SPLINE
SPL {X  -146.983, Y  +302.107, Z    +0.000, E1   +74.473, E3 +78846.478}
SPL {X  -146.624, Y  +301.420, Z    +0.000, E1   +73.294, E3 +78856.962}
SPL {X  -144.830, Y  +298.101, Z    +0.000, E1   +72.333, E3 +78866.485}
SPL {X  -140.483, Y  +290.724, Z    +0.000, E1   +71.922, E3 +78873.643}
SPL {X  -136.362, Y  +284.451, Z    +0.000, E1   +71.514, E3 +78879.809}
SPL {X  -132.604, Y  +279.221, Z    +0.000, E1   +70.988, E3 +78885.838}
SPL {X  -129.663, Y  +275.410, Z    +0.000, E1   +70.632, E3 +78889.761}
SPL {X  -127.149, Y  +272.325, Z    +0.000, E1   +70.073, E3 +78894.141}
SPL {X  -123.924, Y  +268.578, Z    +0.000, E1   +70.633, E3 +78893.958}
SPL {X  -115.163, Y  +259.431, Z    +0.000, E1   +74.058, E3 +78885.067}
SPL {X   -55.479, Y  +222.417, Z    +0.000, E1   +56.403, E3 +79070.921}
ENDSPLINE

SPLINE
SPL {X  -130.757, Y  +276.802, Z    +0.000, E1   +58.343, E3 +79226.857}
SPL {X  -154.788, Y  +319.502, Z    +0.000, E1   +45.389, E3 +79231.056}
SPL {X  -161.887, Y  +343.393, Z    +0.000, E1   +32.461, E3 +79231.512}
SPL {X  -164.949, Y  +363.277, Z    +0.000, E1   +17.059, E3 +79230.787}
SPL {X  -165.638, Y  +376.493, Z    +0.000, E1    +4.395, E3 +79230.425}
SPL {X  -165.650, Y  +380.829, Z    +0.000, E1    -0.360, E3 +79229.405}
SPL {X  -165.650, Y  +385.053, Z    +0.000, E1   -10.073, E3 +79228.913}
SPL {X  -165.650, Y  +388.847, Z    +0.000, E1   -19.524, E3 +79228.878}
SPL {X  -165.650, Y  +394.451, Z    +0.000, E1   -33.170, E3 +79228.291}
SPL {X  -165.650, Y  +401.692, Z    +0.000, E1   -47.300, E3 +79228.273}
SPL {X  -165.650, Y  +412.079, Z    +0.000, E1   -62.360, E3 +79226.115}
SPL {X  -165.650, Y  +422.274, Z    +0.000, E1   -68.953, E3 +79226.601}
SPL {X  -165.650, Y  +470.008, Z    +0.000, E1   -77.011, E3 +79234.818}
SPL {X  -161.095, Y  +714.078, Z    +0.000, E1   -78.221, E3 +79310.354}
ENDSPLINE

SPLINE
SPL {X  -163.418, Y  +702.603, Z    +0.000, E1   -74.313, E3 +79347.749}
ENDSPLINE

SPLINE
SPL {X  -160.284, Y  +717.322, Z    +0.000, E1   -73.988, E3 +79359.513}
SPL {X  -156.453, Y  +729.928, Z    +0.000, E1   -73.507, E3 +79371.665}
SPL {X  -152.193, Y  +740.900, Z    +0.000, E1   -73.135, E3 +79381.232}
SPL {X  -148.880, Y  +748.126, Z    +0.000, E1   -72.716, E3 +79389.013}
SPL {X  -145.823, Y  +754.085, Z    +0.000, E1   -72.288, E3 +79395.784}
SPL {X  -141.906, Y  +760.955, Z    +0.000, E1   -72.057, E3 +79401.475}
SPL {X  -138.580, Y  +766.249, Z    +0.000, E1   -71.449, E3 +79408.565}
SPL {X  -134.851, Y  +771.704, Z    +0.000, E1   -71.081, E3 +79413.960}
SPL {X  -131.668, Y  +776.015, Z    +0.000, E1   -70.566, E3 +79419.234}
SPL {X  -127.547, Y  +781.197, Z    +0.000, E1   -70.083, E3 +79424.597}
SPL {X  -118.977, Y  +790.758, Z    +0.000, E1   -71.976, E3 +79422.115}
SPL {X   -54.368, Y  +831.974, Z    +0.000, E1   -57.152, E3 +79573.904}
ENDSPLINE

SPLINE
SPL {X  -111.514, Y  +797.993, Z    +0.000, E1   -63.064, E3 +79760.035}
SPL {X  -140.675, Y  +762.967, Z    +0.000, E1   -56.489, E3 +79765.998}
SPL {X  -155.138, Y  +733.569, Z    +0.000, E1   -46.550, E3 +79768.302}
SPL {X  -161.585, Y  +711.971, Z    +0.000, E1   -34.503, E3 +79767.352}
SPL {X  -164.796, Y  +692.295, Z    +0.000, E1   -19.289, E3 +79767.387}
SPL {X  -165.632, Y  +677.938, Z    +0.000, E1    -5.073, E3 +79766.758}
SPL {X  -165.650, Y  +673.500, Z    +0.000, E1    +0.000, E3 +79765.792}
SPL {X  -165.650, Y  +671.349, Z    +0.000, E1    +4.619, E3 +79765.297}
SPL {X  -165.650, Y  +666.568, Z    +0.000, E1   +16.799, E3 +79765.172}
SPL {X  -165.650, Y  +661.246, Z    +0.000, E1   +30.569, E3 +79764.952}
SPL {X  -165.650, Y  +652.403, Z    +0.000, E1   +48.665, E3 +79764.591}
SPL {X  -165.650, Y  +637.100, Z    +0.000, E1   +69.106, E3 +79760.931}
SPL {X  -165.650, Y  +616.344, Z    +0.000, E1   +74.941, E3 +79764.181}
SPL {X  -165.650, Y  +575.817, Z    +0.000, E1   +77.800, E3 +79773.110}
SPL {X  -161.405, Y  +341.238, Z    +0.000, E1   +76.606, E3 +79864.409}
SPL {X  -146.302, Y  +300.811, Z    +0.000, E1   +78.008, E3 +79865.526}
ENDSPLINE

SPLINE
SPL {X  -147.825, Y  +303.750, Z    +0.000, E1   +76.548, E3 +79879.958}
SPL {X  -148.167, Y  +304.430, Z    +0.000, E1   +75.276, E3 +79892.051}
ENDSPLINE

SPLINE
SPL {X  -146.983, Y  +302.107, Z    +0.000, E1   +74.473, E3 +79900.532}
SPL {X  -146.624, Y  +301.420, Z    +0.000, E1   +73.294, E3 +79911.016}
SPL {X  -144.830, Y  +298.101, Z    +0.000, E1   +72.333, E3 +79920.540}
SPL {X  -140.483, Y  +290.724, Z    +0.000, E1   +71.922, E3 +79927.697}
SPL {X  -136.362, Y  +284.451, Z    +0.000, E1   +71.514, E3 +79933.863}
SPL {X  -132.604, Y  +279.221, Z    +0.000, E1   +70.988, E3 +79939.892}
SPL {X  -129.663, Y  +275.410, Z    +0.000, E1   +70.632, E3 +79943.815}
SPL {X  -127.149, Y  +272.325, Z    +0.000, E1   +70.073, E3 +79948.195}
SPL {X  -123.924, Y  +268.578, Z    +0.000, E1   +70.633, E3 +79948.012}
SPL {X  -115.163, Y  +259.431, Z    +0.000, E1   +74.058, E3 +79939.121}
SPL {X   -55.479, Y  +222.417, Z    +0.000, E1   +56.403, E3 +80124.975}
ENDSPLINE

SPLINE
SPL {X  -130.757, Y  +276.802, Z    +0.000, E1   +58.343, E3 +80280.911}
SPL {X  -154.788, Y  +319.502, Z    +0.000, E1   +45.389, E3 +80285.110}
SPL {X  -161.887, Y  +343.393, Z    +0.000, E1   +32.461, E3 +80285.566}
SPL {X  -164.949, Y  +363.277, Z    +0.000, E1   +17.059, E3 +80284.841}
SPL {X  -165.638, Y  +376.493, Z    +0.000, E1    +4.395, E3 +80284.479}
SPL {X  -165.650, Y  +380.500, Z    +0.000, E1    +0.000, E3 +80283.590}
SPL {X  -165.650, Y  +381.832, Z    +0.000, E1    -2.686, E3 +80283.062}
SPL {X  -165.650, Y  +385.053, Z    +0.000, E1   -10.073, E3 +80282.967}
SPL {X  -165.650, Y  +388.847, Z    +0.000, E1   -19.524, E3 +80282.932}
SPL {X  -165.650, Y  +393.562, Z    +0.000, E1   -31.212, E3 +80282.415}
SPL {X  -165.650, Y  +400.090, Z    +0.000, E1   -44.561, E3 +80282.270}
SPL {X  -165.650, Y  +415.429, Z    +0.000, E1   -64.815, E3 +80280.329}
SPL {X  -165.650, Y  +470.008, Z    +0.000, E1   -77.011, E3 +80288.873}
SPL {X  -160.882, Y  +714.957, Z    +0.000, E1   -77.470, E3 +80372.578}
ENDSPLINE

SPLINE
SPL {X  -163.522, Y  +701.969, Z    +0.000, E1   -74.236, E3 +80402.234}
ENDSPLINE

SPLINE
SPL {X  -160.284, Y  +717.322, Z    +0.000, E1   -73.988, E3 +80413.567}
SPL {X  -156.453, Y  +729.928, Z    +0.000, E1   -73.507, E3 +80425.719}
SPL {X  -152.193, Y  +740.900, Z    +0.000, E1   -73.135, E3 +80435.286}
SPL {X  -148.880, Y  +748.126, Z    +0.000, E1   -72.716, E3 +80443.067}
SPL {X  -144.434, Y  +756.610, Z    +0.000, E1   -72.338, E3 +80450.917}
SPL {X  -141.532, Y  +761.573, Z    +0.000, E1   -71.800, E3 +80457.557}
SPL {X  -138.580, Y  +766.249, Z    +0.000, E1   -71.449, E3 +80462.619}
SPL {X  -134.851, Y  +771.704, Z    +0.000, E1   -71.081, E3 +80468.014}
SPL {X  -131.668, Y  +776.015, Z    +0.000, E1   -70.566, E3 +80473.288}
SPL {X  -128.114, Y  +780.508, Z    +0.000, E1   -70.155, E3 +80477.883}
SPL {X  -123.825, Y  +785.533, Z    +0.000, E1   -70.642, E3 +80478.631}
SPL {X  -111.068, Y  +798.397, Z    +0.000, E1   -72.944, E3 +80476.075}
SPL {X   -54.135, Y  +832.054, Z    +0.000, E1   -56.519, E3 +80652.094}
ENDSPLINE

SPLINE
SPL {X  -119.915, Y  +789.781, Z    +0.000, E1   -62.637, E3 +80819.710}
SPL {X  -140.675, Y  +762.967, Z    +0.000, E1   -56.489, E3 +80820.052}
SPL {X  -155.138, Y  +733.569, Z    +0.000, E1   -46.550, E3 +80822.356}
SPL {X  -161.585, Y  +711.971, Z    +0.000, E1   -34.503, E3 +80821.407}
SPL {X  -164.796, Y  +692.295, Z    +0.000, E1   -19.289, E3 +80821.441}
SPL {X  -165.632, Y  +677.938, Z    +0.000, E1    -5.073, E3 +80820.812}
SPL {X  -165.650, Y  +673.500, Z    +0.000, E1    +0.000, E3 +80819.846}
SPL {X  -165.650, Y  +671.349, Z    +0.000, E1    +4.619, E3 +80819.351}
SPL {X  -165.650, Y  +666.568, Z    +0.000, E1   +16.799, E3 +80819.226}
SPL {X  -165.650, Y  +661.246, Z    +0.000, E1   +30.569, E3 +80819.007}
SPL {X  -165.650, Y  +652.403, Z    +0.000, E1   +48.665, E3 +80818.645}
SPL {X  -165.650, Y  +637.100, Z    +0.000, E1   +69.106, E3 +80814.985}
SPL {X  -165.650, Y  +616.344, Z    +0.000, E1   +74.941, E3 +80818.235}
SPL {X  -165.650, Y  +575.817, Z    +0.000, E1   +77.800, E3 +80827.164}
SPL {X  -161.405, Y  +341.238, Z    +0.000, E1   +76.606, E3 +80918.463}
SPL {X  -146.302, Y  +300.811, Z    +0.000, E1   +78.008, E3 +80919.580}
ENDSPLINE

SPLINE
SPL {X  -147.825, Y  +303.750, Z    +0.000, E1   +76.548, E3 +80934.013}
SPL {X  -148.167, Y  +304.430, Z    +0.000, E1   +75.276, E3 +80946.105}
ENDSPLINE

SPLINE
SPL {X  -146.983, Y  +302.107, Z    +0.000, E1   +74.473, E3 +80954.586}
SPL {X  -146.624, Y  +301.420, Z    +0.000, E1   +73.294, E3 +80965.070}
SPL {X  -144.830, Y  +298.101, Z    +0.000, E1   +72.333, E3 +80974.594}
SPL {X  -140.980, Y  +291.526, Z    +0.000, E1   +72.160, E3 +80979.519}
SPL {X  -137.379, Y  +285.943, Z    +0.000, E1   +71.537, E3 +80986.973}
SPL {X  -133.329, Y  +280.198, Z    +0.000, E1   +71.389, E3 +80991.002}
SPL {X  -130.835, Y  +276.902, Z    +0.000, E1   +70.642, E3 +80996.998}
SPL {X  -127.149, Y  +272.325, Z    +0.000, E1   +70.073, E3 +81002.249}
SPL {X  -123.924, Y  +268.578, Z    +0.000, E1   +70.633, E3 +81002.066}
SPL {X  -115.163, Y  +259.431, Z    +0.000, E1   +74.058, E3 +80993.175}
SPL {X   -55.479, Y  +222.417, Z    +0.000, E1   +56.403, E3 +81179.029}
ENDSPLINE

SPLINE
SPL {X  -130.757, Y  +276.802, Z    +0.000, E1   +58.343, E3 +81334.966}
SPL {X  -154.788, Y  +319.502, Z    +0.000, E1   +45.389, E3 +81339.164}
SPL {X  -161.887, Y  +343.393, Z    +0.000, E1   +32.461, E3 +81339.620}
SPL {X  -164.949, Y  +363.277, Z    +0.000, E1   +17.059, E3 +81338.895}
SPL {X  -165.638, Y  +376.493, Z    +0.000, E1    +4.395, E3 +81338.534}
SPL {X  -165.650, Y  +380.500, Z    +0.000, E1    +0.000, E3 +81337.644}
SPL {X  -165.650, Y  +381.832, Z    +0.000, E1    -2.686, E3 +81337.116}
SPL {X  -165.650, Y  +385.053, Z    +0.000, E1   -10.073, E3 +81337.021}
SPL {X  -165.650, Y  +388.847, Z    +0.000, E1   -19.524, E3 +81336.986}
SPL {X  -165.650, Y  +393.562, Z    +0.000, E1   -31.212, E3 +81336.470}
SPL {X  -165.650, Y  +400.090, Z    +0.000, E1   -44.561, E3 +81336.324}
SPL {X  -165.650, Y  +415.429, Z    +0.000, E1   -64.815, E3 +81334.383}
SPL {X  -165.650, Y  +470.008, Z    +0.000, E1   -77.011, E3 +81342.927}
SPL {X  -160.882, Y  +714.957, Z    +0.000, E1   -77.470, E3 +81426.632}
ENDSPLINE

SPLINE
SPL {X  -164.302, Y  +696.586, Z    +0.000, E1   -74.218, E3 +81453.294}
ENDSPLINE

SPLINE
SPL {X  -160.977, Y  +714.570, Z    +0.000, E1   -74.086, E3 +81465.206}
SPL {X  -156.453, Y  +729.928, Z    +0.000, E1   -73.507, E3 +81479.773}
SPL {X  -152.193, Y  +740.900, Z    +0.000, E1   -73.135, E3 +81489.340}
SPL {X  -148.880, Y  +748.126, Z    +0.000, E1   -72.716, E3 +81497.121}
SPL {X  -144.434, Y  +756.610, Z    +0.000, E1   -72.338, E3 +81504.971}
SPL {X  -141.532, Y  +761.573, Z    +0.000, E1   -71.800, E3 +81511.611}
SPL {X  -138.580, Y  +766.249, Z    +0.000, E1   -71.449, E3 +81516.673}
SPL {X  -134.851, Y  +771.704, Z    +0.000, E1   -71.081, E3 +81522.068}
SPL {X  -131.668, Y  +776.015, Z    +0.000, E1   -70.566, E3 +81527.342}
SPL {X  -128.114, Y  +780.508, Z    +0.000, E1   -70.155, E3 +81531.937}
SPL {X  -125.843, Y  +783.219, Z    +0.000, E1   -69.779, E3 +81535.041}
SPL {X  -118.977, Y  +790.758, Z    +0.000, E1   -71.976, E3 +81530.223}
SPL {X   -54.135, Y  +832.054, Z    +0.000, E1   -56.519, E3 +81706.148}
ENDSPLINE

SPLINE
SPL {X  -119.915, Y  +789.781, Z    +0.000, E1   -62.637, E3 +81873.764}
SPL {X  -140.675, Y  +762.967, Z    +0.000, E1   -56.489, E3 +81874.106}
SPL {X  -155.138, Y  +733.569, Z    +0.000, E1   -46.550, E3 +81876.410}
SPL {X  -161.585, Y  +711.971, Z    +0.000, E1   -34.503, E3 +81875.461}
SPL {X  -164.796, Y  +692.295, Z    +0.000, E1   -19.289, E3 +81875.495}
SPL {X  -165.571, Y  +680.631, Z    +0.000, E1    -7.833, E3 +81874.942}
SPL {X  -165.650, Y  +673.591, Z    +0.000, E1    -0.194, E3 +81873.946}
SPL {X  -165.650, Y  +671.349, Z    +0.000, E1    +4.619, E3 +81873.405}
SPL {X  -165.650, Y  +666.568, Z    +0.000, E1   +16.799, E3 +81873.281}
SPL {X  -165.650, Y  +661.246, Z    +0.000, E1   +30.569, E3 +81873.061}
SPL {X  -165.650, Y  +655.398, Z    +0.000, E1   +43.871, E3 +81872.508}
SPL {X  -165.650, Y  +646.168, Z    +0.000, E1   +58.442, E3 +81871.603}
SPL {X  -165.650, Y  +629.125, Z    +0.000, E1   +72.389, E3 +81869.900}
SPL {X  -165.650, Y  +575.817, Z    +0.000, E1   +77.800, E3 +81881.218}
SPL {X  -161.405, Y  +341.238, Z    +0.000, E1   +76.606, E3 +81972.518}
SPL {X  -146.302, Y  +300.811, Z    +0.000, E1   +78.008, E3 +81973.634}
ENDSPLINE

SPLINE
SPL {X  -147.825, Y  +303.750, Z    +0.000, E1   +76.548, E3 +81988.067}
SPL {X  -148.167, Y  +304.430, Z    +0.000, E1   +75.276, E3 +82000.159}
ENDSPLINE

SPLINE
SPL {X  -146.983, Y  +302.107, Z    +0.000, E1   +74.473, E3 +82008.640}
SPL {X  -146.624, Y  +301.420, Z    +0.000, E1   +73.294, E3 +82019.124}
SPL {X  -144.830, Y  +298.101, Z    +0.000, E1   +72.333, E3 +82028.648}
SPL {X  -140.980, Y  +291.526, Z    +0.000, E1   +72.160, E3 +82033.573}
SPL {X  -137.379, Y  +285.943, Z    +0.000, E1   +71.537, E3 +82041.028}
SPL {X  -133.329, Y  +280.198, Z    +0.000, E1   +71.389, E3 +82045.056}
SPL {X  -130.835, Y  +276.902, Z    +0.000, E1   +70.642, E3 +82051.052}
SPL {X  -127.149, Y  +272.325, Z    +0.000, E1   +70.073, E3 +82056.303}
SPL {X  -123.924, Y  +268.578, Z    +0.000, E1   +70.633, E3 +82056.120}
SPL {X  -115.163, Y  +259.431, Z    +0.000, E1   +74.058, E3 +82047.229}
SPL {X   -55.479, Y  +222.417, Z    +0.000, E1   +56.403, E3 +82233.083}
ENDSPLINE

SPLINE
SPL {X  -130.757, Y  +276.802, Z    +0.000, E1   +58.343, E3 +82389.020}
SPL {X  -154.788, Y  +319.502, Z    +0.000, E1   +45.389, E3 +82393.218}
SPL {X  -161.887, Y  +343.393, Z    +0.000, E1   +32.461, E3 +82393.674}
SPL {X  -164.949, Y  +363.277, Z    +0.000, E1   +17.059, E3 +82392.949}
SPL {X  -165.638, Y  +376.493, Z    +0.000, E1    +4.395, E3 +82392.588}
SPL {X  -165.650, Y  +380.500, Z    +0.000, E1    +0.000, E3 +82391.698}
SPL {X  -165.650, Y  +381.832, Z    +0.000, E1    -2.686, E3 +82391.170}
SPL {X  -165.650, Y  +385.053, Z    +0.000, E1   -10.073, E3 +82391.075}
SPL {X  -165.650, Y  +388.847, Z    +0.000, E1   -19.524, E3 +82391.040}
SPL {X  -165.650, Y  +393.562, Z    +0.000, E1   -31.212, E3 +82390.524}
SPL {X  -165.650, Y  +400.090, Z    +0.000, E1   -44.561, E3 +82390.378}
SPL {X  -165.650, Y  +415.429, Z    +0.000, E1   -64.815, E3 +82388.437}
SPL {X  -165.650, Y  +470.008, Z    +0.000, E1   -77.011, E3 +82396.981}
SPL {X  -160.882, Y  +714.957, Z    +0.000, E1   -77.470, E3 +82480.687}
ENDSPLINE

SPLINE
SPL {X  -164.302, Y  +696.586, Z    +0.000, E1   -74.218, E3 +82507.348}
ENDSPLINE

SPLINE
SPL {X  -160.977, Y  +714.570, Z    +0.000, E1   -74.086, E3 +82519.260}
SPL {X  -156.453, Y  +729.928, Z    +0.000, E1   -73.507, E3 +82533.827}
SPL {X  -152.193, Y  +740.900, Z    +0.000, E1   -73.135, E3 +82543.394}
SPL {X  -148.880, Y  +748.126, Z    +0.000, E1   -72.716, E3 +82551.175}
SPL {X  -144.434, Y  +756.610, Z    +0.000, E1   -72.338, E3 +82559.025}
SPL {X  -141.532, Y  +761.573, Z    +0.000, E1   -71.800, E3 +82565.665}
SPL {X  -138.580, Y  +766.249, Z    +0.000, E1   -71.449, E3 +82570.727}
SPL {X  -134.851, Y  +771.704, Z    +0.000, E1   -71.081, E3 +82576.122}
SPL {X  -131.668, Y  +776.015, Z    +0.000, E1   -70.566, E3 +82581.396}
SPL {X  -128.114, Y  +780.508, Z    +0.000, E1   -70.155, E3 +82585.991}
SPL {X  -125.843, Y  +783.219, Z    +0.000, E1   -69.779, E3 +82589.095}
SPL {X  -118.977, Y  +790.758, Z    +0.000, E1   -71.976, E3 +82584.277}
SPL {X   -54.135, Y  +832.054, Z    +0.000, E1   -56.519, E3 +82760.202}
ENDSPLINE

SPLINE
SPL {X  -119.915, Y  +789.781, Z    +0.000, E1   -62.637, E3 +82927.818}
SPL {X  -140.675, Y  +762.967, Z    +0.000, E1   -56.489, E3 +82928.160}
SPL {X  -155.138, Y  +733.569, Z    +0.000, E1   -46.550, E3 +82930.464}
SPL {X  -161.585, Y  +711.971, Z    +0.000, E1   -34.503, E3 +82929.515}
SPL {X  -164.796, Y  +692.295, Z    +0.000, E1   -19.289, E3 +82929.549}
SPL {X  -165.571, Y  +680.631, Z    +0.000, E1    -7.833, E3 +82928.996}
SPL {X  -165.650, Y  +673.591, Z    +0.000, E1    -0.194, E3 +82928.000}
SPL {X  -165.650, Y  +671.349, Z    +0.000, E1    +4.619, E3 +82927.459}
SPL {X  -165.650, Y  +666.568, Z    +0.000, E1   +16.799, E3 +82927.335}
SPL {X  -165.650, Y  +661.246, Z    +0.000, E1   +30.569, E3 +82927.115}
SPL {X  -165.650, Y  +655.398, Z    +0.000, E1   +43.871, E3 +82926.562}
SPL {X  -165.650, Y  +646.168, Z    +0.000, E1   +58.442, E3 +82925.657}
SPL {X  -165.650, Y  +629.125, Z    +0.000, E1   +72.389, E3 +82923.954}
SPL {X  -165.650, Y  +575.817, Z    +0.000, E1   +77.800, E3 +82935.272}
SPL {X  -161.405, Y  +341.238, Z    +0.000, E1   +76.606, E3 +83026.572}
SPL {X  -146.302, Y  +300.811, Z    +0.000, E1   +78.008, E3 +83027.688}
ENDSPLINE

SPLINE
SPL {X  -147.825, Y  +303.750, Z    +0.000, E1   +76.548, E3 +83042.121}
SPL {X  -148.167, Y  +304.430, Z    +0.000, E1   +75.276, E3 +83054.214}
ENDSPLINE

SPLINE
SPL {X  -146.983, Y  +302.107, Z    +0.000, E1   +74.473, E3 +83062.694}
SPL {X  -146.624, Y  +301.420, Z    +0.000, E1   +73.294, E3 +83073.178}
SPL {X  -144.830, Y  +298.101, Z    +0.000, E1   +72.333, E3 +83082.702}
SPL {X  -140.980, Y  +291.526, Z    +0.000, E1   +72.160, E3 +83087.627}
SPL {X  -137.379, Y  +285.943, Z    +0.000, E1   +71.537, E3 +83095.082}
SPL {X  -133.329, Y  +280.198, Z    +0.000, E1   +71.389, E3 +83099.110}
SPL {X  -130.835, Y  +276.902, Z    +0.000, E1   +70.642, E3 +83105.106}
SPL {X  -127.149, Y  +272.325, Z    +0.000, E1   +70.073, E3 +83110.358}
SPL {X  -123.924, Y  +268.578, Z    +0.000, E1   +70.633, E3 +83110.174}
SPL {X  -115.163, Y  +259.431, Z    +0.000, E1   +74.058, E3 +83101.284}
SPL {X   -55.479, Y  +222.417, Z    +0.000, E1   +56.403, E3 +83287.137}
ENDSPLINE

SPLINE
SPL {X  -130.757, Y  +276.802, Z    +0.000, E1   +58.343, E3 +83443.074}
SPL {X  -154.788, Y  +319.502, Z    +0.000, E1   +45.389, E3 +83447.272}
SPL {X  -161.887, Y  +343.393, Z    +0.000, E1   +32.461, E3 +83447.728}
SPL {X  -164.949, Y  +363.277, Z    +0.000, E1   +17.059, E3 +83447.003}
SPL {X  -165.638, Y  +376.493, Z    +0.000, E1    +4.395, E3 +83446.642}
SPL {X  -165.650, Y  +380.500, Z    +0.000, E1    +0.000, E3 +83445.752}
SPL {X  -165.650, Y  +381.832, Z    +0.000, E1    -2.686, E3 +83445.224}
SPL {X  -165.650, Y  +385.053, Z    +0.000, E1   -10.073, E3 +83445.129}
SPL {X  -165.650, Y  +388.847, Z    +0.000, E1   -19.524, E3 +83445.094}
SPL {X  -165.650, Y  +393.562, Z    +0.000, E1   -31.212, E3 +83444.578}
SPL {X  -165.650, Y  +400.090, Z    +0.000, E1   -44.561, E3 +83444.432}
SPL {X  -165.650, Y  +415.429, Z    +0.000, E1   -64.815, E3 +83442.491}
SPL {X  -165.650, Y  +470.008, Z    +0.000, E1   -77.011, E3 +83451.035}
SPL {X  -160.882, Y  +714.957, Z    +0.000, E1   -77.470, E3 +83534.741}
ENDSPLINE

SPLINE
SPL {X  -164.302, Y  +696.586, Z    +0.000, E1   -74.218, E3 +83561.403}
ENDSPLINE

SPLINE
SPL {X  -160.977, Y  +714.570, Z    +0.000, E1   -74.086, E3 +83573.314}
SPL {X  -156.453, Y  +729.928, Z    +0.000, E1   -73.507, E3 +83587.881}
SPL {X  -152.193, Y  +740.900, Z    +0.000, E1   -73.135, E3 +83597.448}
SPL {X  -148.880, Y  +748.126, Z    +0.000, E1   -72.716, E3 +83605.229}
SPL {X  -144.434, Y  +756.610, Z    +0.000, E1   -72.338, E3 +83613.079}
SPL {X  -141.532, Y  +761.573, Z    +0.000, E1   -71.800, E3 +83619.719}
SPL {X  -138.580, Y  +766.249, Z    +0.000, E1   -71.449, E3 +83624.781}
SPL {X  -134.851, Y  +771.704, Z    +0.000, E1   -71.081, E3 +83630.176}
SPL {X  -131.668, Y  +776.015, Z    +0.000, E1   -70.566, E3 +83635.450}
SPL {X  -128.114, Y  +780.508, Z    +0.000, E1   -70.155, E3 +83640.045}
SPL {X  -125.843, Y  +783.219, Z    +0.000, E1   -69.779, E3 +83643.149}
SPL {X  -118.977, Y  +790.758, Z    +0.000, E1   -71.976, E3 +83638.331}
SPL {X   -54.135, Y  +832.054, Z    +0.000, E1   -56.519, E3 +83814.256}
ENDSPLINE

SPLINE
SPL {X  -119.915, Y  +789.781, Z    +0.000, E1   -62.637, E3 +83981.872}
SPL {X  -140.675, Y  +762.967, Z    +0.000, E1   -56.489, E3 +83982.214}
SPL {X  -155.138, Y  +733.569, Z    +0.000, E1   -46.550, E3 +83984.519}
SPL {X  -161.585, Y  +711.971, Z    +0.000, E1   -34.503, E3 +83983.569}
SPL {X  -164.796, Y  +692.295, Z    +0.000, E1   -19.289, E3 +83983.603}
SPL {X  -165.571, Y  +680.631, Z    +0.000, E1    -7.833, E3 +83983.050}
SPL {X  -165.650, Y  +673.591, Z    +0.000, E1    -0.194, E3 +83982.054}
SPL {X  -165.650, Y  +671.349, Z    +0.000, E1    +4.619, E3 +83981.513}
SPL {X  -165.650, Y  +666.568, Z    +0.000, E1   +16.799, E3 +83981.389}
SPL {X  -165.650, Y  +661.246, Z    +0.000, E1   +30.569, E3 +83981.169}
SPL {X  -165.650, Y  +655.398, Z    +0.000, E1   +43.871, E3 +83980.616}
SPL {X  -165.650, Y  +646.168, Z    +0.000, E1   +58.442, E3 +83979.711}
SPL {X  -165.650, Y  +629.125, Z    +0.000, E1   +72.389, E3 +83978.008}
SPL {X  -165.650, Y  +575.817, Z    +0.000, E1   +77.800, E3 +83989.326}
SPL {X  -161.405, Y  +341.238, Z    +0.000, E1   +76.606, E3 +84080.626}
SPL {X  -146.302, Y  +300.811, Z    +0.000, E1   +78.008, E3 +84081.742}
ENDSPLINE

SPLINE
SPL {X  -147.825, Y  +303.750, Z    +0.000, E1   +76.548, E3 +84096.175}
SPL {X  -148.167, Y  +304.430, Z    +0.000, E1   +75.276, E3 +84108.268}
ENDSPLINE

SPLINE
SPL {X  -146.983, Y  +302.107, Z    +0.000, E1   +74.473, E3 +84116.748}
SPL {X  -146.624, Y  +301.420, Z    +0.000, E1   +73.294, E3 +84127.232}
SPL {X  -144.830, Y  +298.101, Z    +0.000, E1   +72.333, E3 +84136.756}
SPL {X  -140.980, Y  +291.526, Z    +0.000, E1   +72.160, E3 +84141.681}
SPL {X  -137.379, Y  +285.943, Z    +0.000, E1   +71.537, E3 +84149.136}
SPL {X  -133.329, Y  +280.198, Z    +0.000, E1   +71.389, E3 +84153.164}
SPL {X  -130.835, Y  +276.902, Z    +0.000, E1   +70.642, E3 +84159.160}
SPL {X  -127.149, Y  +272.325, Z    +0.000, E1   +70.073, E3 +84164.412}
SPL {X  -123.924, Y  +268.578, Z    +0.000, E1   +70.633, E3 +84164.228}
SPL {X  -115.163, Y  +259.431, Z    +0.000, E1   +74.058, E3 +84155.338}
SPL {X   -55.479, Y  +222.417, Z    +0.000, E1   +56.403, E3 +84341.191}
ENDSPLINE

SPLINE
SPL {X  -130.757, Y  +276.802, Z    +0.000, E1   +58.343, E3 +84497.128}
SPL {X  -154.788, Y  +319.502, Z    +0.000, E1   +45.389, E3 +84501.326}
SPL {X  -161.887, Y  +343.393, Z    +0.000, E1   +32.461, E3 +84501.782}
SPL {X  -164.949, Y  +363.277, Z    +0.000, E1   +17.059, E3 +84501.057}
SPL {X  -165.638, Y  +376.493, Z    +0.000, E1    +4.395, E3 +84500.696}
SPL {X  -165.650, Y  +380.500, Z    +0.000, E1    +0.000, E3 +84499.806}
SPL {X  -165.650, Y  +381.832, Z    +0.000, E1    -2.686, E3 +84499.278}
SPL {X  -165.650, Y  +385.053, Z    +0.000, E1   -10.073, E3 +84499.183}
SPL {X  -165.650, Y  +388.847, Z    +0.000, E1   -19.524, E3 +84499.148}
SPL {X  -165.650, Y  +393.562, Z    +0.000, E1   -31.212, E3 +84498.632}
SPL {X  -165.650, Y  +400.090, Z    +0.000, E1   -44.561, E3 +84498.486}
SPL {X  -165.650, Y  +415.429, Z    +0.000, E1   -64.815, E3 +84496.545}
SPL {X  -165.650, Y  +470.008, Z    +0.000, E1   -77.011, E3 +84505.089}
SPL {X  -160.882, Y  +714.957, Z    +0.000, E1   -77.470, E3 +84588.795}
ENDSPLINE

SPLINE
SPL {X  -164.302, Y  +696.586, Z    +0.000, E1   -74.218, E3 +84615.457}
ENDSPLINE

SPLINE
SPL {X  -160.977, Y  +714.570, Z    +0.000, E1   -74.086, E3 +84627.368}
SPL {X  -156.453, Y  +729.928, Z    +0.000, E1   -73.507, E3 +84641.935}
SPL {X  -152.193, Y  +740.900, Z    +0.000, E1   -73.135, E3 +84651.502}
SPL {X  -148.880, Y  +748.126, Z    +0.000, E1   -72.716, E3 +84659.283}
SPL {X  -144.434, Y  +756.610, Z    +0.000, E1   -72.338, E3 +84667.133}
SPL {X  -141.532, Y  +761.573, Z    +0.000, E1   -71.800, E3 +84673.773}
SPL {X  -138.580, Y  +766.249, Z    +0.000, E1   -71.449, E3 +84678.835}
SPL {X  -134.851, Y  +771.704, Z    +0.000, E1   -71.081, E3 +84684.230}
SPL {X  -130.513, Y  +777.511, Z    +0.000, E1   -70.561, E3 +84690.413}
SPL {X  -127.002, Y  +781.850, Z    +0.000, E1   -69.819, E3 +84696.268}
SPL {X  -118.977, Y  +790.758, Z    +0.000, E1   -71.976, E3 +84692.385}
SPL {X   -54.368, Y  +831.974, Z    +0.000, E1   -57.152, E3 +84844.174}
ENDSPLINE

SPLINE
SPL {X  -111.514, Y  +797.993, Z    +0.000, E1   -63.064, E3 +85030.305}
SPL {X  -140.675, Y  +762.967, Z    +0.000, E1   -56.489, E3 +85036.268}
SPL {X  -155.138, Y  +733.569, Z    +0.000, E1   -46.550, E3 +85038.573}
SPL {X  -162.699, Y  +706.626, Z    +0.000, E1   -30.890, E3 +85037.614}
SPL {X  -165.076, Y  +689.274, Z    +0.000, E1   -16.447, E3 +85037.702}
SPL {X  -165.632, Y  +677.938, Z    +0.000, E1    -5.073, E3 +85037.028}
SPL {X  -165.650, Y  +673.500, Z    +0.000, E1    +0.000, E3 +85036.063}
SPL {X  -165.650, Y  +671.349, Z    +0.000, E1    +4.619, E3 +85035.567}
SPL {X  -165.650, Y  +666.568, Z    +0.000, E1   +16.799, E3 +85035.443}
SPL {X  -165.650, Y  +661.246, Z    +0.000, E1   +30.569, E3 +85035.223}
SPL {X  -165.650, Y  +652.403, Z    +0.000, E1   +48.665, E3 +85034.861}
SPL {X  -165.650, Y  +637.100, Z    +0.000, E1   +69.106, E3 +85031.201}
SPL {X  -165.650, Y  +616.344, Z    +0.000, E1   +74.941, E3 +85034.451}
SPL {X  -165.650, Y  +575.817, Z    +0.000, E1   +77.800, E3 +85043.380}
SPL {X  -161.405, Y  +341.238, Z    +0.000, E1   +76.606, E3 +85134.680}
SPL {X  -146.302, Y  +300.811, Z    +0.000, E1   +78.008, E3 +85135.797}
ENDSPLINE

SPLINE
SPL {X  -147.825, Y  +303.750, Z    +0.000, E1   +76.548, E3 +85150.229}
SPL {X  -148.167, Y  +304.430, Z    +0.000, E1   +75.276, E3 +85162.322}
ENDSPLINE

SPLINE
SPL {X  -146.983, Y  +302.107, Z    +0.000, E1   +74.473, E3 +85170.802}
SPL {X  -146.624, Y  +301.420, Z    +0.000, E1   +73.294, E3 +85181.286}
SPL {X  -144.830, Y  +298.101, Z    +0.000, E1   +72.333, E3 +85190.810}
SPL {X  -140.980, Y  +291.526, Z    +0.000, E1   +72.160, E3 +85195.735}
SPL {X  -138.254, Y  +287.254, Z    +0.000, E1   +71.707, E3 +85201.221}
SPL {X  -134.627, Y  +281.983, Z    +0.000, E1   +71.294, E3 +85206.746}
SPL {X  -132.106, Y  +278.560, Z    +0.000, E1   +70.638, E3 +85212.269}
SPL {X  -129.663, Y  +275.410, Z    +0.000, E1   +70.632, E3 +85214.086}
SPL {X  -127.149, Y  +272.325, Z    +0.000, E1   +70.073, E3 +85218.466}
SPL {X  -123.924, Y  +268.578, Z    +0.000, E1   +70.633, E3 +85218.282}
SPL {X  -115.163, Y  +259.431, Z    +0.000, E1   +74.058, E3 +85209.392}
SPL {X   -55.479, Y  +222.417, Z    +0.000, E1   +56.403, E3 +85395.245}
ENDSPLINE

SPLINE
SPL {X  -130.757, Y  +276.802, Z    +0.000, E1   +58.343, E3 +85551.182}
SPL {X  -157.227, Y  +326.349, Z    +0.000, E1   +42.092, E3 +85554.827}
SPL {X  -163.771, Y  +353.623, Z    +0.000, E1   +25.144, E3 +85556.040}
SPL {X  -165.462, Y  +370.602, Z    +0.000, E1   +10.342, E3 +85554.990}
SPL {X  -165.650, Y  +380.752, Z    +0.000, E1    -0.182, E3 +85553.770}
SPL {X  -165.650, Y  +385.053, Z    +0.000, E1   -10.073, E3 +85553.237}
SPL {X  -165.650, Y  +388.847, Z    +0.000, E1   -19.524, E3 +85553.202}
SPL {X  -165.650, Y  +393.562, Z    +0.000, E1   -31.212, E3 +85552.686}
SPL {X  -165.650, Y  +400.090, Z    +0.000, E1   -44.561, E3 +85552.540}
SPL {X  -165.650, Y  +415.429, Z    +0.000, E1   -64.815, E3 +85550.599}
SPL {X  -165.650, Y  +460.635, Z    +0.000, E1   -76.744, E3 +85556.496}
SPL {X  -165.650, Y  +476.745, Z    +0.000, E1   -77.150, E3 +85561.048}
SPL {X  -161.095, Y  +714.078, Z    +0.000, E1   -78.221, E3 +85634.678}
ENDSPLINE

SPLINE
SPL {X  -163.418, Y  +702.603, Z    +0.000, E1   -74.313, E3 +85672.074}
ENDSPLINE

SPLINE
SPL {X  -160.284, Y  +717.322, Z    +0.000, E1   -73.988, E3 +85683.837}
SPL {X  -156.453, Y  +729.928, Z    +0.000, E1   -73.507, E3 +85695.989}
SPL {X  -152.193, Y  +740.900, Z    +0.000, E1   -73.135, E3 +85705.556}
SPL {X  -148.880, Y  +748.126, Z    +0.000, E1   -72.716, E3 +85713.337}
SPL {X  -144.434, Y  +756.610, Z    +0.000, E1   -72.338, E3 +85721.187}
SPL {X  -141.532, Y  +761.573, Z    +0.000, E1   -71.800, E3 +85727.827}
SPL {X  -138.580, Y  +766.249, Z    +0.000, E1   -71.449, E3 +85732.889}
SPL {X  -134.851, Y  +771.704, Z    +0.000, E1   -71.081, E3 +85738.284}
SPL {X  -130.513, Y  +777.511, Z    +0.000, E1   -70.561, E3 +85744.467}
SPL {X  -127.002, Y  +781.850, Z    +0.000, E1   -69.819, E3 +85750.322}
SPL {X  -121.778, Y  +787.794, Z    +0.000, E1   -71.623, E3 +85746.370}
SPL {X  -111.068, Y  +798.397, Z    +0.000, E1   -72.944, E3 +85746.346}
SPL {X   -54.368, Y  +831.974, Z    +0.000, E1   -57.152, E3 +85898.228}
ENDSPLINE

SPLINE
SPL {X  -111.514, Y  +797.993, Z    +0.000, E1   -63.064, E3 +86084.359}
SPL {X  -140.675, Y  +762.967, Z    +0.000, E1   -56.489, E3 +86090.322}
SPL {X  -155.138, Y  +733.569, Z    +0.000, E1   -46.550, E3 +86092.627}
SPL {X  -162.699, Y  +706.626, Z    +0.000, E1   -30.890, E3 +86091.668}
SPL {X  -165.420, Y  +684.230, Z    +0.000, E1   -11.665, E3 +86091.419}
SPL {X  -165.650, Y  +673.591, Z    +0.000, E1    -0.194, E3 +86090.162}
SPL {X  -165.650, Y  +671.349, Z    +0.000, E1    +4.619, E3 +86089.621}
SPL {X  -165.650, Y  +666.568, Z    +0.000, E1   +16.799, E3 +86089.497}
SPL {X  -165.650, Y  +661.246, Z    +0.000, E1   +30.569, E3 +86089.277}
SPL {X  -165.650, Y  +655.398, Z    +0.000, E1   +43.871, E3 +86088.724}
SPL {X  -165.650, Y  +648.742, Z    +0.000, E1   +53.940, E3 +86089.148}
SPL {X  -165.650, Y  +637.100, Z    +0.000, E1   +69.106, E3 +86085.255}
SPL {X  -165.650, Y  +616.344, Z    +0.000, E1   +74.941, E3 +86088.505}
SPL {X  -165.650, Y  +575.817, Z    +0.000, E1   +77.800, E3 +86097.434}
SPL {X  -161.405, Y  +341.238, Z    +0.000, E1   +76.606, E3 +86188.734}
SPL {X  -146.302, Y  +300.811, Z    +0.000, E1   +78.008, E3 +86189.851}
ENDSPLINE

SPLINE
SPL {X  -147.825, Y  +303.750, Z    +0.000, E1   +76.548, E3 +86204.283}
SPL {X  -148.167, Y  +304.430, Z    +0.000, E1   +75.276, E3 +86216.376}
ENDSPLINE

SPLINE
SPL {X  -146.983, Y  +302.107, Z    +0.000, E1   +74.473, E3 +86224.856}
SPL {X  -146.624, Y  +301.420, Z    +0.000, E1   +73.294, E3 +86235.340}
SPL {X  -144.830, Y  +298.101, Z    +0.000, E1   +72.333, E3 +86244.864}
SPL {X  -140.980, Y  +291.526, Z    +0.000, E1   +72.160, E3 +86249.789}
SPL {X  -137.379, Y  +285.943, Z    +0.000, E1   +71.537, E3 +86257.244}
SPL {X  -133.329, Y  +280.198, Z    +0.000, E1   +71.389, E3 +86261.272}
SPL {X  -130.835, Y  +276.902, Z    +0.000, E1   +70.642, E3 +86267.268}
SPL {X  -127.149, Y  +272.325, Z    +0.000, E1   +70.073, E3 +86272.520}
SPL {X  -123.924, Y  +268.578, Z    +0.000, E1   +70.633, E3 +86272.336}
SPL {X  -115.163, Y  +259.431, Z    +0.000, E1   +74.058, E3 +86263.446}
SPL {X   -55.479, Y  +222.417, Z    +0.000, E1   +56.403, E3 +86449.299}
ENDSPLINE

SPLINE
SPL {X  -130.757, Y  +276.802, Z    +0.000, E1   +58.343, E3 +86605.236}
SPL {X  -157.227, Y  +326.349, Z    +0.000, E1   +42.092, E3 +86608.881}
SPL {X  -163.771, Y  +353.623, Z    +0.000, E1   +25.144, E3 +86610.094}
SPL {X  -165.171, Y  +365.918, Z    +0.000, E1   +14.637, E3 +86609.308}
SPL {X  -165.638, Y  +376.493, Z    +0.000, E1    +4.395, E3 +86608.804}
SPL {X  -165.650, Y  +380.500, Z    +0.000, E1    +0.000, E3 +86607.914}
SPL {X  -165.650, Y  +381.832, Z    +0.000, E1    -2.686, E3 +86607.386}
SPL {X  -165.650, Y  +385.053, Z    +0.000, E1   -10.073, E3 +86607.291}
SPL {X  -165.650, Y  +388.847, Z    +0.000, E1   -19.524, E3 +86607.256}
SPL {X  -165.650, Y  +393.562, Z    +0.000, E1   -31.212, E3 +86606.740}
SPL {X  -165.650, Y  +400.090, Z    +0.000, E1   -44.561, E3 +86606.594}
SPL {X  -165.650, Y  +415.429, Z    +0.000, E1   -64.815, E3 +86604.653}
SPL {X  -165.650, Y  +470.008, Z    +0.000, E1   -77.011, E3 +86613.197}
SPL {X  -160.882, Y  +714.957, Z    +0.000, E1   -77.470, E3 +86696.903}
ENDSPLINE

SPLINE
SPL {X  -164.302, Y  +696.586, Z    +0.000, E1   -74.218, E3 +86723.565}
ENDSPLINE

SPLINE
SPL {X  -160.977, Y  +714.570, Z    +0.000, E1   -74.086, E3 +86735.476}
SPL {X  -156.453, Y  +729.928, Z    +0.000, E1   -73.507, E3 +86750.044}
SPL {X  -152.193, Y  +740.900, Z    +0.000, E1   -73.135, E3 +86759.610}
SPL {X  -148.880, Y  +748.126, Z    +0.000, E1   -72.716, E3 +86767.391}
SPL {X  -145.823, Y  +754.085, Z    +0.000, E1   -72.288, E3 +86774.163}
SPL {X  -141.906, Y  +760.955, Z    +0.000, E1   -72.057, E3 +86779.853}
SPL {X  -138.580, Y  +766.249, Z    +0.000, E1   -71.449, E3 +86786.943}
SPL {X  -134.851, Y  +771.704, Z    +0.000, E1   -71.081, E3 +86792.338}
SPL {X  -131.668, Y  +776.015, Z    +0.000, E1   -70.566, E3 +86797.612}
SPL {X  -127.547, Y  +781.197, Z    +0.000, E1   -70.083, E3 +86802.976}
SPL {X  -118.977, Y  +790.758, Z    +0.000, E1   -71.976, E3 +86800.493}
SPL {X   -54.135, Y  +832.054, Z    +0.000, E1   -56.519, E3 +86976.419}
ENDSPLINE

SPLINE
SPL {X  -119.915, Y  +789.781, Z    +0.000, E1   -62.637, E3 +87144.034}
SPL {X  -140.675, Y  +762.967, Z    +0.000, E1   -56.489, E3 +87144.376}
SPL {X  -155.138, Y  +733.569, Z    +0.000, E1   -46.550, E3 +87146.681}
SPL {X  -161.585, Y  +711.971, Z    +0.000, E1   -34.503, E3 +87145.731}
SPL {X  -164.796, Y  +692.295, Z    +0.000, E1   -19.289, E3 +87145.765}
SPL {X  -165.632, Y  +677.938, Z    +0.000, E1    -5.073, E3 +87145.136}
SPL {X  -165.650, Y  +673.500, Z    +0.000, E1    +0.000, E3 +87144.171}
SPL {X  -165.650, Y  +671.349, Z    +0.000, E1    +4.619, E3 +87143.675}
SPL {X  -165.650, Y  +666.568, Z    +0.000, E1   +16.799, E3 +87143.551}
SPL {X  -165.650, Y  +661.246, Z    +0.000, E1   +30.569, E3 +87143.331}
SPL {X  -165.650, Y  +652.403, Z    +0.000, E1   +48.665, E3 +87142.969}
SPL {X  -165.650, Y  +637.100, Z    +0.000, E1   +69.106, E3 +87139.309}
SPL {X  -165.650, Y  +616.344, Z    +0.000, E1   +74.941, E3 +87142.559}
SPL {X  -165.650, Y  +575.817, Z    +0.000, E1   +77.800, E3 +87151.488}
SPL {X  -161.405, Y  +341.238, Z    +0.000, E1   +76.606, E3 +87242.788}
SPL {X  -146.302, Y  +300.811, Z    +0.000, E1   +78.008, E3 +87243.905}
ENDSPLINE

SPLINE
SPL {X  -147.825, Y  +303.750, Z    +0.000, E1   +76.548, E3 +87258.337}
SPL {X  -148.167, Y  +304.430, Z    +0.000, E1   +75.276, E3 +87270.430}
ENDSPLINE

SPLINE
SPL {X  -146.983, Y  +302.107, Z    +0.000, E1   +74.473, E3 +87278.910}
SPL {X  -146.624, Y  +301.420, Z    +0.000, E1   +73.294, E3 +87289.394}
SPL {X  -144.830, Y  +298.101, Z    +0.000, E1   +72.333, E3 +87298.918}
SPL {X  -140.980, Y  +291.526, Z    +0.000, E1   +72.160, E3 +87303.843}
SPL {X  -137.379, Y  +285.943, Z    +0.000, E1   +71.537, E3 +87311.298}
SPL {X  -133.329, Y  +280.198, Z    +0.000, E1   +71.389, E3 +87315.326}
SPL {X  -130.835, Y  +276.902, Z    +0.000, E1   +70.642, E3 +87321.322}
SPL {X  -127.149, Y  +272.325, Z    +0.000, E1   +70.073, E3 +87326.574}
SPL {X  -123.924, Y  +268.578, Z    +0.000, E1   +70.633, E3 +87326.390}
SPL {X  -115.163, Y  +259.431, Z    +0.000, E1   +74.058, E3 +87317.500}
SPL {X   -55.479, Y  +222.417, Z    +0.000, E1   +56.403, E3 +87503.354}
ENDSPLINE

SPLINE
SPL {X  -130.757, Y  +276.802, Z    +0.000, E1   +58.343, E3 +87659.290}
SPL {X  -157.227, Y  +326.349, Z    +0.000, E1   +42.092, E3 +87662.936}
SPL {X  -163.771, Y  +353.623, Z    +0.000, E1   +25.144, E3 +87664.148}
SPL {X  -165.171, Y  +365.918, Z    +0.000, E1   +14.637, E3 +87663.362}
SPL {X  -165.638, Y  +376.493, Z    +0.000, E1    +4.395, E3 +87662.858}
SPL {X  -165.650, Y  +380.500, Z    +0.000, E1    +0.000, E3 +87661.968}
SPL {X  -165.650, Y  +381.832, Z    +0.000, E1    -2.686, E3 +87661.440}
SPL {X  -165.650, Y  +385.053, Z    +0.000, E1   -10.073, E3 +87661.345}
SPL {X  -165.650, Y  +388.847, Z    +0.000, E1   -19.524, E3 +87661.310}
SPL {X  -165.650, Y  +393.562, Z    +0.000, E1   -31.212, E3 +87660.794}
SPL {X  -165.650, Y  +400.090, Z    +0.000, E1   -44.561, E3 +87660.648}
SPL {X  -165.650, Y  +415.429, Z    +0.000, E1   -64.815, E3 +87658.707}
SPL {X  -165.650, Y  +470.008, Z    +0.000, E1   -77.011, E3 +87667.251}
SPL {X  -160.882, Y  +714.957, Z    +0.000, E1   -77.470, E3 +87750.957}
ENDSPLINE

SPLINE
SPL {X  -164.302, Y  +696.586, Z    +0.000, E1   -74.218, E3 +87777.619}
ENDSPLINE

SPLINE
SPL {X  -160.977, Y  +714.570, Z    +0.000, E1   -74.086, E3 +87789.530}
SPL {X  -156.453, Y  +729.928, Z    +0.000, E1   -73.507, E3 +87804.098}
SPL {X  -152.193, Y  +740.900, Z    +0.000, E1   -73.135, E3 +87813.664}
SPL {X  -148.880, Y  +748.126, Z    +0.000, E1   -72.716, E3 +87821.445}
SPL {X  -145.823, Y  +754.085, Z    +0.000, E1   -72.288, E3 +87828.217}
SPL {X  -141.906, Y  +760.955, Z    +0.000, E1   -72.057, E3 +87833.907}
SPL {X  -138.580, Y  +766.249, Z    +0.000, E1   -71.449, E3 +87840.997}
SPL {X  -134.851, Y  +771.704, Z    +0.000, E1   -71.081, E3 +87846.392}
SPL {X  -131.668, Y  +776.015, Z    +0.000, E1   -70.566, E3 +87851.666}
SPL {X  -127.547, Y  +781.197, Z    +0.000, E1   -70.083, E3 +87857.030}
SPL {X  -118.977, Y  +790.758, Z    +0.000, E1   -71.976, E3 +87854.547}
SPL {X   -54.368, Y  +831.974, Z    +0.000, E1   -57.152, E3 +88006.336}
ENDSPLINE

SPLINE
SPL {X  -111.514, Y  +797.993, Z    +0.000, E1   -63.064, E3 +88192.467}
SPL {X  -140.675, Y  +762.967, Z    +0.000, E1   -56.489, E3 +88198.430}
SPL {X  -155.138, Y  +733.569, Z    +0.000, E1   -46.550, E3 +88200.735}
SPL {X  -162.699, Y  +706.626, Z    +0.000, E1   -30.890, E3 +88199.776}
SPL {X  -165.076, Y  +689.274, Z    +0.000, E1   -16.447, E3 +88199.864}
SPL {X  -165.632, Y  +677.938, Z    +0.000, E1    -5.073, E3 +88199.191}
SPL {X  -165.650, Y  +673.297, Z    +0.000, E1    +0.232, E3 +88198.147}
SPL {X  -165.650, Y  +670.223, Z    +0.000, E1    +7.575, E3 +88197.628}
SPL {X  -165.650, Y  +666.568, Z    +0.000, E1   +16.799, E3 +88197.605}
SPL {X  -165.650, Y  +661.246, Z    +0.000, E1   +30.569, E3 +88197.385}
SPL {X  -165.650, Y  +652.403, Z    +0.000, E1   +48.665, E3 +88197.023}
SPL {X  -165.650, Y  +637.100, Z    +0.000, E1   +69.106, E3 +88193.363}
SPL {X  -165.650, Y  +616.344, Z    +0.000, E1   +74.941, E3 +88196.613}
SPL {X  -165.650, Y  +575.817, Z    +0.000, E1   +77.800, E3 +88205.542}
SPL {X  -162.613, Y  +346.923, Z    +0.000, E1   +78.263, E3 +88277.215}
SPL {X  -161.207, Y  +340.393, Z    +0.000, E1   +75.705, E3 +88307.078}
SPL {X  -146.302, Y  +300.811, Z    +0.000, E1   +78.008, E3 +88297.959}
ENDSPLINE

SPLINE
SPL {X  -147.825, Y  +303.750, Z    +0.000, E1   +76.548, E3 +88312.391}
SPL {X  -148.167, Y  +304.430, Z    +0.000, E1   +75.276, E3 +88324.484}
ENDSPLINE

SPLINE
SPL {X  -146.983, Y  +302.107, Z    +0.000, E1   +74.473, E3 +88332.965}
SPL {X  -146.624, Y  +301.420, Z    +0.000, E1   +73.294, E3 +88343.448}
SPL {X  -144.830, Y  +298.101, Z    +0.000, E1   +72.333, E3 +88352.972}
SPL {X  -140.980, Y  +291.526, Z    +0.000, E1   +72.160, E3 +88357.897}
SPL {X  -137.379, Y  +285.943, Z    +0.000, E1   +71.537, E3 +88365.352}
SPL {X  -133.329, Y  +280.198, Z    +0.000, E1   +71.389, E3 +88369.380}
SPL {X  -130.835, Y  +276.902, Z    +0.000, E1   +70.642, E3 +88375.376}
SPL {X  -127.149, Y  +272.325, Z    +0.000, E1   +70.073, E3 +88380.628}
SPL {X  -123.924, Y  +268.578, Z    +0.000, E1   +70.633, E3 +88380.444}
SPL {X  -115.163, Y  +259.431, Z    +0.000, E1   +74.058, E3 +88371.554}
SPL {X   -55.479, Y  +222.417, Z    +0.000, E1   +56.403, E3 +88557.408}
ENDSPLINE

SPLINE
SPL {X  -130.757, Y  +276.802, Z    +0.000, E1   +58.343, E3 +88713.344}
SPL {X  -157.227, Y  +326.349, Z    +0.000, E1   +42.092, E3 +88716.990}
SPL {X  -163.771, Y  +353.623, Z    +0.000, E1   +25.144, E3 +88718.202}
SPL {X  -165.171, Y  +365.918, Z    +0.000, E1   +14.637, E3 +88717.416}
SPL {X  -165.638, Y  +376.493, Z    +0.000, E1    +4.395, E3 +88716.912}
SPL {X  -165.650, Y  +380.829, Z    +0.000, E1    -0.360, E3 +88715.892}
SPL {X  -165.650, Y  +385.053, Z    +0.000, E1   -10.073, E3 +88715.400}
SPL {X  -165.650, Y  +388.847, Z    +0.000, E1   -19.524, E3 +88715.364}
SPL {X  -165.650, Y  +393.562, Z    +0.000, E1   -31.212, E3 +88714.848}
SPL {X  -165.650, Y  +400.090, Z    +0.000, E1   -44.561, E3 +88714.702}
SPL {X  -165.650, Y  +415.429, Z    +0.000, E1   -64.815, E3 +88712.761}
SPL {X  -165.650, Y  +470.008, Z    +0.000, E1   -77.011, E3 +88721.305}
SPL {X  -160.882, Y  +714.957, Z    +0.000, E1   -77.470, E3 +88805.011}
ENDSPLINE

SPLINE
SPL {X  -164.302, Y  +696.586, Z    +0.000, E1   -74.218, E3 +88831.673}
ENDSPLINE

SPLINE
SPL {X  -160.977, Y  +714.570, Z    +0.000, E1   -74.086, E3 +88843.584}
SPL {X  -156.453, Y  +729.928, Z    +0.000, E1   -73.507, E3 +88858.152}
SPL {X  -152.193, Y  +740.900, Z    +0.000, E1   -73.135, E3 +88867.718}
SPL {X  -148.880, Y  +748.126, Z    +0.000, E1   -72.716, E3 +88875.499}
SPL {X  -145.823, Y  +754.085, Z    +0.000, E1   -72.288, E3 +88882.271}
SPL {X  -141.906, Y  +760.955, Z    +0.000, E1   -72.057, E3 +88887.961}
SPL {X  -138.580, Y  +766.249, Z    +0.000, E1   -71.449, E3 +88895.051}
SPL {X  -134.851, Y  +771.704, Z    +0.000, E1   -71.081, E3 +88900.446}
SPL {X  -130.513, Y  +777.511, Z    +0.000, E1   -70.561, E3 +88906.629}
SPL {X  -127.002, Y  +781.850, Z    +0.000, E1   -69.819, E3 +88912.484}
SPL {X  -118.977, Y  +790.758, Z    +0.000, E1   -71.976, E3 +88908.601}
SPL {X   -54.368, Y  +831.974, Z    +0.000, E1   -57.152, E3 +89060.390}
ENDSPLINE

SPLINE
SPL {X  -111.514, Y  +797.993, Z    +0.000, E1   -63.064, E3 +89246.521}
SPL {X  -140.675, Y  +762.967, Z    +0.000, E1   -56.489, E3 +89252.484}
SPL {X  -155.138, Y  +733.569, Z    +0.000, E1   -46.550, E3 +89254.789}
SPL {X  -162.699, Y  +706.626, Z    +0.000, E1   -30.890, E3 +89253.830}
SPL {X  -165.076, Y  +689.274, Z    +0.000, E1   -16.447, E3 +89253.918}
SPL {X  -165.632, Y  +677.938, Z    +0.000, E1    -5.073, E3 +89253.245}
SPL {X  -165.650, Y  +673.297, Z    +0.000, E1    +0.232, E3 +89252.201}
SPL {X  -165.650, Y  +670.223, Z    +0.000, E1    +7.575, E3 +89251.682}
SPL {X  -165.650, Y  +666.568, Z    +0.000, E1   +16.799, E3 +89251.659}
SPL {X  -165.650, Y  +661.246, Z    +0.000, E1   +30.569, E3 +89251.439}
SPL {X  -165.650, Y  +652.403, Z    +0.000, E1   +48.665, E3 +89251.077}
SPL {X  -165.650, Y  +637.100, Z    +0.000, E1   +69.106, E3 +89247.417}
SPL {X  -165.650, Y  +616.344, Z    +0.000, E1   +74.941, E3 +89250.667}
SPL {X  -165.650, Y  +575.817, Z    +0.000, E1   +77.800, E3 +89259.596}
SPL {X  -162.613, Y  +346.923, Z    +0.000, E1   +78.263, E3 +89331.269}
SPL {X  -161.207, Y  +340.393, Z    +0.000, E1   +75.705, E3 +89361.132}
SPL {X  -146.302, Y  +300.811, Z    +0.000, E1   +78.008, E3 +89352.013}
ENDSPLINE

SPLINE
SPL {X  -147.825, Y  +303.750, Z    +0.000, E1   +76.548, E3 +89366.445}
SPL {X  -148.167, Y  +304.430, Z    +0.000, E1   +75.276, E3 +89378.538}
ENDSPLINE

SPLINE
SPL {X  -146.983, Y  +302.107, Z    +0.000, E1   +74.473, E3 +89387.019}
SPL {X  -146.624, Y  +301.420, Z    +0.000, E1   +73.294, E3 +89397.502}
SPL {X  -144.830, Y  +298.101, Z    +0.000, E1   +72.333, E3 +89407.026}
SPL {X  -140.980, Y  +291.526, Z    +0.000, E1   +72.160, E3 +89411.951}
SPL {X  -137.379, Y  +285.943, Z    +0.000, E1   +71.537, E3 +89419.406}
SPL {X  -133.329, Y  +280.198, Z    +0.000, E1   +71.389, E3 +89423.434}
SPL {X  -130.835, Y  +276.902, Z    +0.000, E1   +70.642, E3 +89429.431}
SPL {X  -127.149, Y  +272.325, Z    +0.000, E1   +70.073, E3 +89434.682}
SPL {X  -123.924, Y  +268.578, Z    +0.000, E1   +70.633, E3 +89434.498}
SPL {X  -115.163, Y  +259.431, Z    +0.000, E1   +74.058, E3 +89425.608}
SPL {X   -55.479, Y  +222.417, Z    +0.000, E1   +56.403, E3 +89611.462}
ENDSPLINE

SPLINE
SPL {X  -130.757, Y  +276.802, Z    +0.000, E1   +58.343, E3 +89767.398}
SPL {X  -157.227, Y  +326.349, Z    +0.000, E1   +42.092, E3 +89771.044}
SPL {X  -163.771, Y  +353.623, Z    +0.000, E1   +25.144, E3 +89772.256}
SPL {X  -165.171, Y  +365.918, Z    +0.000, E1   +14.637, E3 +89771.470}
SPL {X  -165.638, Y  +376.493, Z    +0.000, E1    +4.395, E3 +89770.966}
SPL {X  -165.650, Y  +380.829, Z    +0.000, E1    -0.360, E3 +89769.946}
SPL {X  -165.650, Y  +385.053, Z    +0.000, E1   -10.073, E3 +89769.454}
SPL {X  -165.650, Y  +388.847, Z    +0.000, E1   -19.524, E3 +89769.418}
SPL {X  -165.650, Y  +393.562, Z    +0.000, E1   -31.212, E3 +89768.902}
SPL {X  -165.650, Y  +400.090, Z    +0.000, E1   -44.561, E3 +89768.756}
SPL {X  -165.650, Y  +415.429, Z    +0.000, E1   -64.815, E3 +89766.815}
SPL {X  -165.650, Y  +470.008, Z    +0.000, E1   -77.011, E3 +89775.359}
SPL {X  -160.882, Y  +714.957, Z    +0.000, E1   -77.470, E3 +89859.065}
ENDSPLINE

SPLINE
SPL {X  -164.302, Y  +696.586, Z    +0.000, E1   -74.218, E3 +89885.727}
ENDSPLINE

SPLINE
SPL {X  -160.977, Y  +714.570, Z    +0.000, E1   -74.086, E3 +89897.638}
SPL {X  -156.453, Y  +729.928, Z    +0.000, E1   -73.507, E3 +89912.206}
SPL {X  -152.193, Y  +740.900, Z    +0.000, E1   -73.135, E3 +89921.772}
SPL {X  -148.880, Y  +748.126, Z    +0.000, E1   -72.716, E3 +89929.553}
SPL {X  -145.823, Y  +754.085, Z    +0.000, E1   -72.288, E3 +89936.325}
SPL {X  -141.906, Y  +760.955, Z    +0.000, E1   -72.057, E3 +89942.015}
SPL {X  -138.580, Y  +766.249, Z    +0.000, E1   -71.449, E3 +89949.105}
SPL {X  -134.851, Y  +771.704, Z    +0.000, E1   -71.081, E3 +89954.501}
SPL {X  -130.513, Y  +777.511, Z    +0.000, E1   -70.561, E3 +89960.683}
SPL {X  -127.002, Y  +781.850, Z    +0.000, E1   -69.819, E3 +89966.538}
SPL {X  -118.977, Y  +790.758, Z    +0.000, E1   -71.976, E3 +89962.655}
SPL {X   -54.135, Y  +832.054, Z    +0.000, E1   -56.519, E3 +90138.581}
ENDSPLINE

SPLINE
SPL {X  -119.915, Y  +789.781, Z    +0.000, E1   -62.637, E3 +90306.196}
SPL {X  -140.675, Y  +762.967, Z    +0.000, E1   -56.489, E3 +90306.538}
SPL {X  -155.138, Y  +733.569, Z    +0.000, E1   -46.550, E3 +90308.843}
SPL {X  -161.585, Y  +711.971, Z    +0.000, E1   -34.503, E3 +90307.893}
SPL {X  -164.796, Y  +692.295, Z    +0.000, E1   -19.289, E3 +90307.928}
SPL {X  -165.632, Y  +677.938, Z    +0.000, E1    -5.073, E3 +90307.299}
SPL {X  -165.650, Y  +673.297, Z    +0.000, E1    +0.232, E3 +90306.255}
SPL {X  -165.650, Y  +670.223, Z    +0.000, E1    +7.575, E3 +90305.736}
SPL {X  -165.650, Y  +666.568, Z    +0.000, E1   +16.799, E3 +90305.713}
SPL {X  -165.650, Y  +661.246, Z    +0.000, E1   +30.569, E3 +90305.493}
SPL {X  -165.650, Y  +655.398, Z    +0.000, E1   +43.871, E3 +90304.941}
SPL {X  -165.650, Y  +646.168, Z    +0.000, E1   +58.442, E3 +90304.036}
SPL {X  -165.650, Y  +629.125, Z    +0.000, E1   +72.389, E3 +90302.332}
SPL {X  -165.650, Y  +575.817, Z    +0.000, E1   +77.800, E3 +90313.650}
SPL {X  -161.405, Y  +341.238, Z    +0.000, E1   +76.606, E3 +90404.950}
SPL {X  -146.302, Y  +300.811, Z    +0.000, E1   +78.008, E3 +90406.067}
ENDSPLINE

SPLINE
SPL {X  -147.825, Y  +303.750, Z    +0.000, E1   +76.548, E3 +90420.499}
SPL {X  -148.167, Y  +304.430, Z    +0.000, E1   +75.276, E3 +90432.592}
ENDSPLINE

SPLINE
SPL {X  -146.983, Y  +302.107, Z    +0.000, E1   +74.473, E3 +90441.073}
SPL {X  -146.624, Y  +301.420, Z    +0.000, E1   +73.294, E3 +90451.556}
SPL {X  -144.830, Y  +298.101, Z    +0.000, E1   +72.333, E3 +90461.080}
SPL {X  -140.980, Y  +291.526, Z    +0.000, E1   +72.160, E3 +90466.005}
SPL {X  -137.379, Y  +285.943, Z    +0.000, E1   +71.537, E3 +90473.460}
SPL {X  -133.329, Y  +280.198, Z    +0.000, E1   +71.389, E3 +90477.488}
SPL {X  -130.835, Y  +276.902, Z    +0.000, E1   +70.642, E3 +90483.485}
SPL {X  -127.149, Y  +272.325, Z    +0.000, E1   +70.073, E3 +90488.736}
SPL {X  -123.924, Y  +268.578, Z    +0.000, E1   +70.633, E3 +90488.552}
SPL {X  -115.163, Y  +259.431, Z    +0.000, E1   +74.058, E3 +90479.662}
SPL {X   -55.479, Y  +222.417, Z    +0.000, E1   +56.403, E3 +90665.516}
ENDSPLINE

SPLINE
SPL {X  -130.757, Y  +276.802, Z    +0.000, E1   +58.343, E3 +90821.452}
SPL {X  -157.227, Y  +326.349, Z    +0.000, E1   +42.092, E3 +90825.098}
SPL {X  -163.771, Y  +353.623, Z    +0.000, E1   +25.144, E3 +90826.311}
SPL {X  -165.462, Y  +370.602, Z    +0.000, E1   +10.342, E3 +90825.260}
SPL {X  -165.650, Y  +380.417, Z    +0.000, E1    +0.167, E3 +90824.176}
SPL {X  -165.650, Y  +381.832, Z    +0.000, E1    -2.686, E3 +90823.602}
SPL {X  -165.650, Y  +385.053, Z    +0.000, E1   -10.073, E3 +90823.508}
SPL {X  -165.650, Y  +388.847, Z    +0.000, E1   -19.524, E3 +90823.472}
SPL {X  -165.650, Y  +393.562, Z    +0.000, E1   -31.212, E3 +90822.956}
SPL {X  -165.650, Y  +400.090, Z    +0.000, E1   -44.561, E3 +90822.810}
SPL {X  -165.650, Y  +415.429, Z    +0.000, E1   -64.815, E3 +90820.869}
SPL {X  -165.650, Y  +460.635, Z    +0.000, E1   -76.744, E3 +90826.766}
SPL {X  -165.650, Y  +476.745, Z    +0.000, E1   -77.150, E3 +90831.318}
SPL {X  -161.095, Y  +714.078, Z    +0.000, E1   -78.221, E3 +90904.948}
ENDSPLINE

SPLINE
SPL {X  -163.418, Y  +702.603, Z    +0.000, E1   -74.313, E3 +90942.344}
ENDSPLINE

SPLINE
SPL {X  -160.284, Y  +717.322, Z    +0.000, E1   -73.988, E3 +90954.108}
SPL {X  -157.512, Y  +726.783, Z    +0.000, E1   -73.653, E3 +90962.821}
SPL {X  -155.383, Y  +732.911, Z    +0.000, E1   -73.297, E3 +90969.748}
SPL {X  -152.193, Y  +740.900, Z    +0.000, E1   -73.135, E3 +90975.826}
SPL {X  -148.880, Y  +748.126, Z    +0.000, E1   -72.716, E3 +90983.608}
SPL {X  -145.823, Y  +754.085, Z    +0.000, E1   -72.288, E3 +90990.379}
SPL {X  -141.906, Y  +760.955, Z    +0.000, E1   -72.057, E3 +90996.070}
SPL {X  -138.580, Y  +766.249, Z    +0.000, E1   -71.449, E3 +91003.159}
SPL {X  -134.851, Y  +771.704, Z    +0.000, E1   -71.081, E3 +91008.555}
SPL {X  -130.513, Y  +777.511, Z    +0.000, E1   -70.561, E3 +91014.737}
SPL {X  -127.002, Y  +781.850, Z    +0.000, E1   -69.819, E3 +91020.592}
SPL {X  -118.977, Y  +790.758, Z    +0.000, E1   -71.976, E3 +91016.709}
SPL {X   -54.135, Y  +832.054, Z    +0.000, E1   -56.519, E3 +91192.635}
ENDSPLINE

SPLINE
SPL {X  -119.915, Y  +789.781, Z    +0.000, E1   -62.637, E3 +91360.250}
SPL {X  -140.675, Y  +762.967, Z    +0.000, E1   -56.489, E3 +91360.592}
SPL {X  -155.138, Y  +733.569, Z    +0.000, E1   -46.550, E3 +91362.897}
SPL {X  -161.585, Y  +711.971, Z    +0.000, E1   -34.503, E3 +91361.947}
SPL {X  -164.796, Y  +692.295, Z    +0.000, E1   -19.289, E3 +91361.982}
SPL {X  -165.632, Y  +677.938, Z    +0.000, E1    -5.073, E3 +91361.353}
SPL {X  -165.650, Y  +673.297, Z    +0.000, E1    +0.232, E3 +91360.309}
SPL {X  -165.650, Y  +670.223, Z    +0.000, E1    +7.575, E3 +91359.790}
SPL {X  -165.650, Y  +666.568, Z    +0.000, E1   +16.799, E3 +91359.767}
SPL {X  -165.650, Y  +661.246, Z    +0.000, E1   +30.569, E3 +91359.547}
SPL {X  -165.650, Y  +655.398, Z    +0.000, E1   +43.871, E3 +91358.995}
SPL {X  -165.650, Y  +646.168, Z    +0.000, E1   +58.442, E3 +91358.090}
SPL {X  -165.650, Y  +629.125, Z    +0.000, E1   +72.389, E3 +91356.386}
SPL {X  -165.650, Y  +575.817, Z    +0.000, E1   +77.800, E3 +91367.704}
SPL {X  -161.405, Y  +341.238, Z    +0.000, E1   +76.606, E3 +91459.004}
SPL {X  -146.302, Y  +300.811, Z    +0.000, E1   +78.008, E3 +91460.121}
ENDSPLINE

SPLINE
SPL {X  -147.825, Y  +303.750, Z    +0.000, E1   +76.548, E3 +91474.553}
SPL {X  -148.167, Y  +304.430, Z    +0.000, E1   +75.276, E3 +91486.646}
ENDSPLINE

SPLINE
SPL {X  -146.983, Y  +302.107, Z    +0.000, E1   +74.473, E3 +91495.127}
SPL {X  -146.624, Y  +301.420, Z    +0.000, E1   +73.294, E3 +91505.610}
SPL {X  -144.830, Y  +298.101, Z    +0.000, E1   +72.333, E3 +91515.134}
SPL {X  -140.483, Y  +290.724, Z    +0.000, E1   +71.922, E3 +91522.291}
SPL {X  -136.362, Y  +284.451, Z    +0.000, E1   +71.514, E3 +91528.458}
SPL {X  -133.329, Y  +280.198, Z    +0.000, E1   +71.389, E3 +91531.543}
SPL {X  -130.835, Y  +276.902, Z    +0.000, E1   +70.642, E3 +91537.539}
SPL {X  -127.149, Y  +272.325, Z    +0.000, E1   +70.073, E3 +91542.790}
SPL {X  -123.924, Y  +268.578, Z    +0.000, E1   +70.633, E3 +91542.606}
SPL {X  -115.163, Y  +259.431, Z    +0.000, E1   +74.058, E3 +91533.716}
SPL {X   -55.479, Y  +222.417, Z    +0.000, E1   +56.403, E3 +91719.570}
ENDSPLINE

SPLINE
SPL {X  -130.757, Y  +276.802, Z    +0.000, E1   +58.343, E3 +91875.506}
SPL {X  -154.788, Y  +319.502, Z    +0.000, E1   +45.389, E3 +91879.705}
SPL {X  -161.887, Y  +343.393, Z    +0.000, E1   +32.461, E3 +91880.161}
SPL {X  -164.949, Y  +363.277, Z    +0.000, E1   +17.059, E3 +91879.436}
SPL {X  -165.638, Y  +376.493, Z    +0.000, E1    +4.395, E3 +91879.074}
SPL {X  -165.650, Y  +380.500, Z    +0.000, E1    +0.000, E3 +91878.184}
SPL {X  -165.650, Y  +381.832, Z    +0.000, E1    -2.686, E3 +91877.656}
SPL {X  -165.650, Y  +385.053, Z    +0.000, E1   -10.073, E3 +91877.562}
SPL {X  -165.650, Y  +388.847, Z    +0.000, E1   -19.524, E3 +91877.526}
SPL {X  -165.650, Y  +393.562, Z    +0.000, E1   -31.212, E3 +91877.010}
SPL {X  -165.650, Y  +400.090, Z    +0.000, E1   -44.561, E3 +91876.864}
SPL {X  -165.650, Y  +415.429, Z    +0.000, E1   -64.815, E3 +91874.923}
SPL {X  -165.650, Y  +470.008, Z    +0.000, E1   -77.011, E3 +91883.467}
SPL {X  -161.095, Y  +714.078, Z    +0.000, E1   -78.221, E3 +91959.002}
ENDSPLINE

SPLINE
SPL {X  -163.418, Y  +702.603, Z    +0.000, E1   -74.313, E3 +91996.398}
ENDSPLINE

SPLINE
SPL {X  -160.284, Y  +717.322, Z    +0.000, E1   -73.988, E3 +92008.162}
SPL {X  -156.453, Y  +729.928, Z    +0.000, E1   -73.507, E3 +92020.314}
SPL {X  -152.193, Y  +740.900, Z    +0.000, E1   -73.135, E3 +92029.880}
SPL {X  -148.880, Y  +748.126, Z    +0.000, E1   -72.716, E3 +92037.662}
SPL {X  -145.823, Y  +754.085, Z    +0.000, E1   -72.288, E3 +92044.433}
SPL {X  -141.906, Y  +760.955, Z    +0.000, E1   -72.057, E3 +92050.124}
SPL {X  -138.580, Y  +766.249, Z    +0.000, E1   -71.449, E3 +92057.213}
SPL {X  -134.851, Y  +771.704, Z    +0.000, E1   -71.081, E3 +92062.609}
SPL {X  -131.668, Y  +776.015, Z    +0.000, E1   -70.566, E3 +92067.882}
SPL {X  -128.114, Y  +780.508, Z    +0.000, E1   -70.155, E3 +92072.478}
SPL {X  -123.825, Y  +785.533, Z    +0.000, E1   -70.642, E3 +92073.226}
SPL {X  -111.068, Y  +798.397, Z    +0.000, E1   -72.944, E3 +92070.670}
SPL {X   -54.135, Y  +832.054, Z    +0.000, E1   -56.519, E3 +92246.689}
ENDSPLINE

SPLINE
SPL {X  -119.915, Y  +789.781, Z    +0.000, E1   -62.637, E3 +92414.304}
SPL {X  -140.675, Y  +762.967, Z    +0.000, E1   -56.489, E3 +92414.646}
SPL {X  -155.138, Y  +733.569, Z    +0.000, E1   -46.550, E3 +92416.951}
SPL {X  -161.585, Y  +711.971, Z    +0.000, E1   -34.503, E3 +92416.001}
SPL {X  -164.796, Y  +692.295, Z    +0.000, E1   -19.289, E3 +92416.036}
SPL {X  -165.632, Y  +677.938, Z    +0.000, E1    -5.073, E3 +92415.407}
SPL {X  -165.650, Y  +673.500, Z    +0.000, E1    +0.000, E3 +92414.441}
SPL {X  -165.650, Y  +671.349, Z    +0.000, E1    +4.619, E3 +92413.945}
SPL {X  -165.650, Y  +666.568, Z    +0.000, E1   +16.799, E3 +92413.821}
SPL {X  -165.650, Y  +661.246, Z    +0.000, E1   +30.569, E3 +92413.601}
SPL {X  -165.650, Y  +652.403, Z    +0.000, E1   +48.665, E3 +92413.239}
SPL {X  -165.650, Y  +637.100, Z    +0.000, E1   +69.106, E3 +92409.579}
SPL {X  -165.650, Y  +616.344, Z    +0.000, E1   +74.941, E3 +92412.829}
SPL {X  -165.650, Y  +575.817, Z    +0.000, E1   +77.800, E3 +92421.758}
SPL {X  -161.405, Y  +341.238, Z    +0.000, E1   +76.606, E3 +92513.058}
SPL {X  -146.302, Y  +300.811, Z    +0.000, E1   +78.008, E3 +92514.175}
ENDSPLINE

SPLINE
SPL {X  -147.825, Y  +303.750, Z    +0.000, E1   +76.548, E3 +92528.607}
SPL {X  -148.167, Y  +304.430, Z    +0.000, E1   +75.276, E3 +92540.700}
ENDSPLINE

SPLINE
SPL {X  -146.983, Y  +302.107, Z    +0.000, E1   +74.473, E3 +92549.181}
SPL {X  -146.624, Y  +301.420, Z    +0.000, E1   +73.294, E3 +92559.665}
SPL {X  -144.830, Y  +298.101, Z    +0.000, E1   +72.333, E3 +92569.188}
SPL {X  -140.980, Y  +291.526, Z    +0.000, E1   +72.160, E3 +92574.113}
SPL {X  -137.379, Y  +285.943, Z    +0.000, E1   +71.537, E3 +92581.568}
SPL {X  -133.329, Y  +280.198, Z    +0.000, E1   +71.389, E3 +92585.597}
SPL {X  -130.835, Y  +276.902, Z    +0.000, E1   +70.642, E3 +92591.593}
SPL {X  -127.149, Y  +272.325, Z    +0.000, E1   +70.073, E3 +92596.844}
SPL {X  -123.924, Y  +268.578, Z    +0.000, E1   +70.633, E3 +92596.660}
SPL {X  -115.163, Y  +259.431, Z    +0.000, E1   +74.058, E3 +92587.770}
SPL {X   -55.479, Y  +222.417, Z    +0.000, E1   +56.403, E3 +92773.624}
ENDSPLINE

SPLINE
SPL {X  -130.757, Y  +276.802, Z    +0.000, E1   +58.343, E3 +92929.560}
SPL {X  -154.788, Y  +319.502, Z    +0.000, E1   +45.389, E3 +92933.759}
SPL {X  -161.887, Y  +343.393, Z    +0.000, E1   +32.461, E3 +92934.215}
SPL {X  -164.949, Y  +363.277, Z    +0.000, E1   +17.059, E3 +92933.490}
SPL {X  -165.638, Y  +376.493, Z    +0.000, E1    +4.395, E3 +92933.128}
SPL {X  -165.650, Y  +380.500, Z    +0.000, E1    +0.000, E3 +92932.238}
SPL {X  -165.650, Y  +381.832, Z    +0.000, E1    -2.686, E3 +92931.710}
SPL {X  -165.650, Y  +385.053, Z    +0.000, E1   -10.073, E3 +92931.616}
SPL {X  -165.650, Y  +388.847, Z    +0.000, E1   -19.524, E3 +92931.580}
SPL {X  -165.650, Y  +393.562, Z    +0.000, E1   -31.212, E3 +92931.064}
SPL {X  -165.650, Y  +400.090, Z    +0.000, E1   -44.561, E3 +92930.919}
SPL {X  -165.650, Y  +415.429, Z    +0.000, E1   -64.815, E3 +92928.977}
SPL {X  -165.650, Y  +470.008, Z    +0.000, E1   -77.011, E3 +92937.521}
SPL {X  -160.882, Y  +714.957, Z    +0.000, E1   -77.470, E3 +93021.227}
ENDSPLINE

SPLINE
SPL {X  -164.302, Y  +696.586, Z    +0.000, E1   -74.218, E3 +93047.889}
ENDSPLINE

SPLINE
SPL {X  -160.977, Y  +714.570, Z    +0.000, E1   -74.086, E3 +93059.800}
SPL {X  -156.453, Y  +729.928, Z    +0.000, E1   -73.507, E3 +93074.368}
SPL {X  -152.193, Y  +740.900, Z    +0.000, E1   -73.135, E3 +93083.934}
SPL {X  -148.880, Y  +748.126, Z    +0.000, E1   -72.716, E3 +93091.716}
SPL {X  -145.823, Y  +754.085, Z    +0.000, E1   -72.288, E3 +93098.487}
SPL {X  -141.906, Y  +760.955, Z    +0.000, E1   -72.057, E3 +93104.178}
SPL {X  -138.580, Y  +766.249, Z    +0.000, E1   -71.449, E3 +93111.268}
SPL {X  -134.851, Y  +771.704, Z    +0.000, E1   -71.081, E3 +93116.663}
SPL {X  -131.668, Y  +776.015, Z    +0.000, E1   -70.566, E3 +93121.936}
SPL {X  -128.114, Y  +780.508, Z    +0.000, E1   -70.155, E3 +93126.532}
SPL {X  -123.825, Y  +785.533, Z    +0.000, E1   -70.642, E3 +93127.280}
SPL {X  -111.068, Y  +798.397, Z    +0.000, E1   -72.944, E3 +93124.724}
SPL {X   -54.368, Y  +831.974, Z    +0.000, E1   -57.152, E3 +93276.607}
ENDSPLINE

SPLINE
SPL {X  -111.514, Y  +797.993, Z    +0.000, E1   -63.064, E3 +93462.738}
SPL {X  -140.675, Y  +762.967, Z    +0.000, E1   -56.489, E3 +93468.700}
SPL {X  -155.138, Y  +733.569, Z    +0.000, E1   -46.550, E3 +93471.005}
SPL {X  -161.585, Y  +711.971, Z    +0.000, E1   -34.503, E3 +93470.055}
SPL {X  -164.796, Y  +692.295, Z    +0.000, E1   -19.289, E3 +93470.090}
SPL {X  -165.632, Y  +677.938, Z    +0.000, E1    -5.073, E3 +93469.461}
SPL {X  -165.650, Y  +673.500, Z    +0.000, E1    +0.000, E3 +93468.495}
SPL {X  -165.650, Y  +671.349, Z    +0.000, E1    +4.619, E3 +93467.999}
SPL {X  -165.650, Y  +666.568, Z    +0.000, E1   +16.799, E3 +93467.875}
SPL {X  -165.650, Y  +661.246, Z    +0.000, E1   +30.569, E3 +93467.655}
SPL {X  -165.650, Y  +652.403, Z    +0.000, E1   +48.665, E3 +93467.293}
SPL {X  -165.650, Y  +637.100, Z    +0.000, E1   +69.106, E3 +93463.633}
SPL {X  -165.650, Y  +616.344, Z    +0.000, E1   +74.941, E3 +93466.883}
SPL {X  -165.650, Y  +575.817, Z    +0.000, E1   +77.800, E3 +93475.812}
SPL {X  -161.405, Y  +341.238, Z    +0.000, E1   +76.606, E3 +93567.112}
SPL {X  -146.302, Y  +300.811, Z    +0.000, E1   +78.008, E3 +93568.229}
ENDSPLINE

SPLINE
SPL {X  -147.825, Y  +303.750, Z    +0.000, E1   +76.548, E3 +93582.661}
SPL {X  -148.167, Y  +304.430, Z    +0.000, E1   +75.276, E3 +93594.754}
ENDSPLINE

SPLINE
SPL {X  -146.983, Y  +302.107, Z    +0.000, E1   +74.473, E3 +93603.235}
SPL {X  -146.624, Y  +301.420, Z    +0.000, E1   +73.294, E3 +93613.719}
SPL {X  -144.830, Y  +298.101, Z    +0.000, E1   +72.333, E3 +93623.242}
SPL {X  -140.483, Y  +290.724, Z    +0.000, E1   +71.922, E3 +93630.399}
SPL {X  -135.200, Y  +282.788, Z    +0.000, E1   +71.482, E3 +93637.745}
SPL {X  -130.835, Y  +276.902, Z    +0.000, E1   +70.642, E3 +93645.647}
SPL {X  -127.149, Y  +272.325, Z    +0.000, E1   +70.073, E3 +93650.898}
SPL {X  -123.924, Y  +268.578, Z    +0.000, E1   +70.633, E3 +93650.714}
SPL {X  -115.163, Y  +259.431, Z    +0.000, E1   +74.058, E3 +93641.824}
SPL {X   -55.479, Y  +222.417, Z    +0.000, E1   +56.403, E3 +93827.678}
ENDSPLINE

SPLINE
SPL {X  -130.757, Y  +276.802, Z    +0.000, E1   +58.343, E3 +93983.614}
SPL {X  -157.227, Y  +326.349, Z    +0.000, E1   +42.092, E3 +93987.260}
SPL {X  -163.771, Y  +353.623, Z    +0.000, E1   +25.144, E3 +93988.473}
SPL {X  -165.171, Y  +365.918, Z    +0.000, E1   +14.637, E3 +93987.687}
SPL {X  -165.638, Y  +376.493, Z    +0.000, E1    +4.395, E3 +93987.182}
SPL {X  -165.650, Y  +380.829, Z    +0.000, E1    -0.360, E3 +93986.162}
SPL {X  -165.650, Y  +385.053, Z    +0.000, E1   -10.073, E3 +93985.670}
SPL {X  -165.650, Y  +388.847, Z    +0.000, E1   -19.524, E3 +93985.634}
SPL {X  -165.650, Y  +393.562, Z    +0.000, E1   -31.212, E3 +93985.118}
SPL {X  -165.650, Y  +400.090, Z    +0.000, E1   -44.561, E3 +93984.973}
SPL {X  -165.650, Y  +415.429, Z    +0.000, E1   -64.815, E3 +93983.031}
SPL {X  -165.650, Y  +460.635, Z    +0.000, E1   -76.744, E3 +93988.928}
SPL {X  -165.650, Y  +476.745, Z    +0.000, E1   -77.150, E3 +93993.480}
SPL {X  -161.095, Y  +714.078, Z    +0.000, E1   -78.221, E3 +94067.110}
ENDSPLINE

SPLINE
SPL {X  -163.418, Y  +702.603, Z    +0.000, E1   -74.313, E3 +94104.506}
ENDSPLINE

SPLINE
SPL {X  -160.284, Y  +717.322, Z    +0.000, E1   -73.988, E3 +94116.270}
SPL {X  -156.453, Y  +729.928, Z    +0.000, E1   -73.507, E3 +94128.422}
SPL {X  -152.193, Y  +740.900, Z    +0.000, E1   -73.135, E3 +94137.988}
SPL {X  -148.880, Y  +748.126, Z    +0.000, E1   -72.716, E3 +94145.770}
SPL {X  -144.434, Y  +756.610, Z    +0.000, E1   -72.338, E3 +94153.620}
SPL {X  -141.532, Y  +761.573, Z    +0.000, E1   -71.800, E3 +94160.260}
SPL {X  -138.580, Y  +766.249, Z    +0.000, E1   -71.449, E3 +94165.322}
SPL {X  -134.851, Y  +771.704, Z    +0.000, E1   -71.081, E3 +94170.717}
SPL {X  -130.513, Y  +777.511, Z    +0.000, E1   -70.561, E3 +94176.899}
SPL {X  -127.002, Y  +781.850, Z    +0.000, E1   -69.819, E3 +94182.754}
SPL {X  -121.778, Y  +787.794, Z    +0.000, E1   -71.623, E3 +94178.802}
SPL {X  -111.068, Y  +798.397, Z    +0.000, E1   -72.944, E3 +94178.778}
SPL {X   -54.368, Y  +831.974, Z    +0.000, E1   -57.152, E3 +94330.661}
ENDSPLINE

SPLINE
SPL {X  -111.514, Y  +797.993, Z    +0.000, E1   -63.064, E3 +94516.792}
SPL {X  -140.675, Y  +762.967, Z    +0.000, E1   -56.489, E3 +94522.754}
SPL {X  -155.138, Y  +733.569, Z    +0.000, E1   -46.550, E3 +94525.059}
SPL {X  -162.699, Y  +706.626, Z    +0.000, E1   -30.890, E3 +94524.101}
SPL {X  -165.420, Y  +684.230, Z    +0.000, E1   -11.665, E3 +94523.852}
SPL {X  -165.650, Y  +673.591, Z    +0.000, E1    -0.194, E3 +94522.595}
SPL {X  -165.650, Y  +671.349, Z    +0.000, E1    +4.619, E3 +94522.053}
SPL {X  -165.650, Y  +666.568, Z    +0.000, E1   +16.799, E3 +94521.929}
SPL {X  -165.650, Y  +661.246, Z    +0.000, E1   +30.569, E3 +94521.709}
SPL {X  -165.650, Y  +655.398, Z    +0.000, E1   +43.871, E3 +94521.157}
SPL {X  -165.650, Y  +648.742, Z    +0.000, E1   +53.940, E3 +94521.580}
SPL {X  -165.650, Y  +637.100, Z    +0.000, E1   +69.106, E3 +94517.687}
SPL {X  -165.650, Y  +616.344, Z    +0.000, E1   +74.941, E3 +94520.937}
SPL {X  -165.650, Y  +575.817, Z    +0.000, E1   +77.800, E3 +94529.866}
SPL {X  -161.405, Y  +341.238, Z    +0.000, E1   +76.606, E3 +94621.166}
SPL {X  -146.302, Y  +300.811, Z    +0.000, E1   +78.008, E3 +94622.283}
ENDSPLINE

SPLINE
SPL {X  -147.825, Y  +303.750, Z    +0.000, E1   +76.548, E3 +94636.715}
SPL {X  -148.167, Y  +304.430, Z    +0.000, E1   +75.276, E3 +94648.808}
ENDSPLINE

SPLINE
SPL {X  -146.983, Y  +302.107, Z    +0.000, E1   +74.473, E3 +94657.289}
SPL {X  -146.624, Y  +301.420, Z    +0.000, E1   +73.294, E3 +94667.773}
SPL {X  -144.830, Y  +298.101, Z    +0.000, E1   +72.333, E3 +94677.296}
SPL {X  -140.980, Y  +291.526, Z    +0.000, E1   +72.160, E3 +94682.222}
SPL {X  -137.379, Y  +285.943, Z    +0.000, E1   +71.537, E3 +94689.676}
SPL {X  -133.329, Y  +280.198, Z    +0.000, E1   +71.389, E3 +94693.705}
SPL {X  -130.835, Y  +276.902, Z    +0.000, E1   +70.642, E3 +94699.701}
SPL {X  -127.149, Y  +272.325, Z    +0.000, E1   +70.073, E3 +94704.952}
SPL {X  -123.924, Y  +268.578, Z    +0.000, E1   +70.633, E3 +94704.768}
SPL {X  -115.163, Y  +259.431, Z    +0.000, E1   +74.058, E3 +94695.878}
SPL {X   -55.479, Y  +222.417, Z    +0.000, E1   +56.403, E3 +94881.732}
ENDSPLINE

SPLINE
SPL {X  -130.757, Y  +276.802, Z    +0.000, E1   +58.343, E3 +95037.668}
SPL {X  -157.227, Y  +326.349, Z    +0.000, E1   +42.092, E3 +95041.314}
SPL {X  -163.771, Y  +353.623, Z    +0.000, E1   +25.144, E3 +95042.527}
SPL {X  -165.171, Y  +365.918, Z    +0.000, E1   +14.637, E3 +95041.741}
SPL {X  -165.638, Y  +376.493, Z    +0.000, E1    +4.395, E3 +95041.236}
SPL {X  -165.650, Y  +380.500, Z    +0.000, E1    +0.000, E3 +95040.346}
SPL {X  -165.650, Y  +381.832, Z    +0.000, E1    -2.686, E3 +95039.818}
SPL {X  -165.650, Y  +385.053, Z    +0.000, E1   -10.073, E3 +95039.724}
SPL {X  -165.650, Y  +388.847, Z    +0.000, E1   -19.524, E3 +95039.688}
SPL {X  -165.650, Y  +393.562, Z    +0.000, E1   -31.212, E3 +95039.172}
SPL {X  -165.650, Y  +400.090, Z    +0.000, E1   -44.561, E3 +95039.027}
SPL {X  -165.650, Y  +415.429, Z    +0.000, E1   -64.815, E3 +95037.085}
SPL {X  -165.650, Y  +470.008, Z    +0.000, E1   -77.011, E3 +95045.629}
SPL {X  -160.882, Y  +714.957, Z    +0.000, E1   -77.470, E3 +95129.335}
ENDSPLINE

SPLINE
SPL {X  -164.302, Y  +696.586, Z    +0.000, E1   -74.218, E3 +95155.997}
ENDSPLINE

SPLINE
SPL {X  -160.977, Y  +714.570, Z    +0.000, E1   -74.086, E3 +95167.909}
SPL {X  -156.453, Y  +729.928, Z    +0.000, E1   -73.507, E3 +95182.476}
SPL {X  -152.193, Y  +740.900, Z    +0.000, E1   -73.135, E3 +95192.042}
SPL {X  -148.880, Y  +748.126, Z    +0.000, E1   -72.716, E3 +95199.824}
SPL {X  -145.823, Y  +754.085, Z    +0.000, E1   -72.288, E3 +95206.595}
SPL {X  -141.906, Y  +760.955, Z    +0.000, E1   -72.057, E3 +95212.286}
SPL {X  -138.580, Y  +766.249, Z    +0.000, E1   -71.449, E3 +95219.376}
SPL {X  -134.851, Y  +771.704, Z    +0.000, E1   -71.081, E3 +95224.771}
SPL {X  -131.668, Y  +776.015, Z    +0.000, E1   -70.566, E3 +95230.044}
SPL {X  -127.547, Y  +781.197, Z    +0.000, E1   -70.083, E3 +95235.408}
SPL {X  -118.977, Y  +790.758, Z    +0.000, E1   -71.976, E3 +95232.926}
SPL {X   -54.135, Y  +832.054, Z    +0.000, E1   -56.519, E3 +95408.851}
ENDSPLINE

SPLINE
SPL {X  -119.915, Y  +789.781, Z    +0.000, E1   -62.637, E3 +95576.466}
SPL {X  -140.675, Y  +762.967, Z    +0.000, E1   -56.489, E3 +95576.809}
SPL {X  -155.138, Y  +733.569, Z    +0.000, E1   -46.550, E3 +95579.113}
SPL {X  -161.585, Y  +711.971, Z    +0.000, E1   -34.503, E3 +95578.163}
SPL {X  -164.796, Y  +692.295, Z    +0.000, E1   -19.289, E3 +95578.198}
SPL {X  -165.632, Y  +677.938, Z    +0.000, E1    -5.073, E3 +95577.569}
SPL {X  -165.650, Y  +673.500, Z    +0.000, E1    +0.000, E3 +95576.603}
SPL {X  -165.650, Y  +671.349, Z    +0.000, E1    +4.619, E3 +95576.107}
SPL {X  -165.650, Y  +666.568, Z    +0.000, E1   +16.799, E3 +95575.983}
SPL {X  -165.650, Y  +661.246, Z    +0.000, E1   +30.569, E3 +95575.763}
SPL {X  -165.650, Y  +652.403, Z    +0.000, E1   +48.665, E3 +95575.401}
SPL {X  -165.650, Y  +637.100, Z    +0.000, E1   +69.106, E3 +95571.741}
SPL {X  -165.650, Y  +616.344, Z    +0.000, E1   +74.941, E3 +95574.991}
SPL {X  -165.650, Y  +575.817, Z    +0.000, E1   +77.800, E3 +95583.920}
SPL {X  -161.405, Y  +341.238, Z    +0.000, E1   +76.606, E3 +95675.220}
SPL {X  -146.302, Y  +300.811, Z    +0.000, E1   +78.008, E3 +95676.337}
ENDSPLINE

SPLINE
SPL {X  -147.825, Y  +303.750, Z    +0.000, E1   +76.548, E3 +95690.769}
SPL {X  -148.167, Y  +304.430, Z    +0.000, E1   +75.276, E3 +95702.862}
ENDSPLINE

SPLINE
SPL {X  -146.983, Y  +302.107, Z    +0.000, E1   +74.473, E3 +95711.343}
SPL {X  -146.624, Y  +301.420, Z    +0.000, E1   +73.294, E3 +95721.827}
SPL {X  -144.830, Y  +298.101, Z    +0.000, E1   +72.333, E3 +95731.350}
SPL {X  -140.980, Y  +291.526, Z    +0.000, E1   +72.160, E3 +95736.276}
SPL {X  -137.379, Y  +285.943, Z    +0.000, E1   +71.537, E3 +95743.730}
SPL {X  -133.329, Y  +280.198, Z    +0.000, E1   +71.389, E3 +95747.759}
SPL {X  -130.835, Y  +276.902, Z    +0.000, E1   +70.642, E3 +95753.755}
SPL {X  -127.149, Y  +272.325, Z    +0.000, E1   +70.073, E3 +95759.006}
SPL {X  -123.924, Y  +268.578, Z    +0.000, E1   +70.633, E3 +95758.822}
SPL {X  -115.163, Y  +259.431, Z    +0.000, E1   +74.058, E3 +95749.932}
SPL {X   -55.479, Y  +222.417, Z    +0.000, E1   +56.403, E3 +95935.786}
ENDSPLINE

SPLINE
SPL {X  -130.757, Y  +276.802, Z    +0.000, E1   +58.343, E3 +96091.722}
SPL {X  -157.227, Y  +326.349, Z    +0.000, E1   +42.092, E3 +96095.368}
SPL {X  -163.771, Y  +353.623, Z    +0.000, E1   +25.144, E3 +96096.581}
SPL {X  -165.171, Y  +365.918, Z    +0.000, E1   +14.637, E3 +96095.795}
SPL {X  -165.638, Y  +376.493, Z    +0.000, E1    +4.395, E3 +96095.290}
SPL {X  -165.650, Y  +380.500, Z    +0.000, E1    +0.000, E3 +96094.400}
SPL {X  -165.650, Y  +381.832, Z    +0.000, E1    -2.686, E3 +96093.872}
SPL {X  -165.650, Y  +385.053, Z    +0.000, E1   -10.073, E3 +96093.778}
SPL {X  -165.650, Y  +388.847, Z    +0.000, E1   -19.524, E3 +96093.742}
SPL {X  -165.650, Y  +393.562, Z    +0.000, E1   -31.212, E3 +96093.226}
SPL {X  -165.650, Y  +400.090, Z    +0.000, E1   -44.561, E3 +96093.081}
SPL {X  -165.650, Y  +415.429, Z    +0.000, E1   -64.815, E3 +96091.139}
SPL {X  -165.650, Y  +470.008, Z    +0.000, E1   -77.011, E3 +96099.683}
SPL {X  -160.882, Y  +714.957, Z    +0.000, E1   -77.470, E3 +96183.389}
ENDSPLINE

SPLINE
SPL {X  -164.302, Y  +696.586, Z    +0.000, E1   -74.218, E3 +96210.051}
ENDSPLINE

SPLINE
SPL {X  -160.977, Y  +714.570, Z    +0.000, E1   -74.086, E3 +96221.963}
SPL {X  -156.453, Y  +729.928, Z    +0.000, E1   -73.507, E3 +96236.530}
SPL {X  -152.193, Y  +740.900, Z    +0.000, E1   -73.135, E3 +96246.096}
SPL {X  -148.880, Y  +748.126, Z    +0.000, E1   -72.716, E3 +96253.878}
SPL {X  -145.823, Y  +754.085, Z    +0.000, E1   -72.288, E3 +96260.649}
SPL {X  -141.906, Y  +760.955, Z    +0.000, E1   -72.057, E3 +96266.340}
SPL {X  -138.580, Y  +766.249, Z    +0.000, E1   -71.449, E3 +96273.430}
SPL {X  -134.851, Y  +771.704, Z    +0.000, E1   -71.081, E3 +96278.825}
SPL {X  -131.668, Y  +776.015, Z    +0.000, E1   -70.566, E3 +96284.098}
SPL {X  -127.547, Y  +781.197, Z    +0.000, E1   -70.083, E3 +96289.462}
SPL {X  -118.977, Y  +790.758, Z    +0.000, E1   -71.976, E3 +96286.980}
SPL {X   -54.135, Y  +832.054, Z    +0.000, E1   -56.519, E3 +96462.905}
ENDSPLINE

SPLINE
SPL {X  -119.915, Y  +789.781, Z    +0.000, E1   -62.637, E3 +96630.520}
SPL {X  -140.675, Y  +762.967, Z    +0.000, E1   -56.489, E3 +96630.863}
SPL {X  -155.138, Y  +733.569, Z    +0.000, E1   -46.550, E3 +96633.167}
SPL {X  -161.585, Y  +711.971, Z    +0.000, E1   -34.503, E3 +96632.217}
SPL {X  -164.796, Y  +692.295, Z    +0.000, E1   -19.289, E3 +96632.252}
SPL {X  -165.632, Y  +677.938, Z    +0.000, E1    -5.073, E3 +96631.623}
SPL {X  -165.650, Y  +673.297, Z    +0.000, E1    +0.232, E3 +96630.580}
SPL {X  -165.650, Y  +670.223, Z    +0.000, E1    +7.575, E3 +96630.060}
SPL {X  -165.650, Y  +666.568, Z    +0.000, E1   +16.799, E3 +96630.037}
SPL {X  -165.650, Y  +661.246, Z    +0.000, E1   +30.569, E3 +96629.817}
SPL {X  -165.650, Y  +655.398, Z    +0.000, E1   +43.871, E3 +96629.265}
SPL {X  -165.650, Y  +646.168, Z    +0.000, E1   +58.442, E3 +96628.360}
SPL {X  -165.650, Y  +629.125, Z    +0.000, E1   +72.389, E3 +96626.656}
SPL {X  -165.650, Y  +575.817, Z    +0.000, E1   +77.800, E3 +96637.974}
SPL {X  -161.405, Y  +341.238, Z    +0.000, E1   +76.606, E3 +96729.274}
SPL {X  -146.302, Y  +300.811, Z    +0.000, E1   +78.008, E3 +96730.391}
ENDSPLINE

SPLINE
SPL {X  -147.825, Y  +303.750, Z    +0.000, E1   +76.548, E3 +96744.823}
SPL {X  -148.167, Y  +304.430, Z    +0.000, E1   +75.276, E3 +96756.916}
ENDSPLINE

SPLINE
SPL {X  -146.983, Y  +302.107, Z    +0.000, E1   +74.473, E3 +96765.397}
SPL {X  -146.624, Y  +301.420, Z    +0.000, E1   +73.294, E3 +96775.881}
SPL {X  -144.830, Y  +298.101, Z    +0.000, E1   +72.333, E3 +96785.404}
SPL {X  -140.980, Y  +291.526, Z    +0.000, E1   +72.160, E3 +96790.330}
SPL {X  -137.379, Y  +285.943, Z    +0.000, E1   +71.537, E3 +96797.784}
SPL {X  -133.329, Y  +280.198, Z    +0.000, E1   +71.389, E3 +96801.813}
SPL {X  -130.835, Y  +276.902, Z    +0.000, E1   +70.642, E3 +96807.809}
SPL {X  -127.149, Y  +272.325, Z    +0.000, E1   +70.073, E3 +96813.060}
SPL {X  -123.924, Y  +268.578, Z    +0.000, E1   +70.633, E3 +96812.876}
SPL {X  -115.163, Y  +259.431, Z    +0.000, E1   +74.058, E3 +96803.986}
SPL {X   -55.479, Y  +222.417, Z    +0.000, E1   +56.403, E3 +96989.840}
ENDSPLINE

SPLINE
SPL {X  -130.757, Y  +276.802, Z    +0.000, E1   +58.343, E3 +97145.776}
SPL {X  -154.788, Y  +319.502, Z    +0.000, E1   +45.389, E3 +97149.975}
SPL {X  -162.966, Y  +348.801, Z    +0.000, E1   +28.734, E3 +97150.059}
SPL {X  -165.462, Y  +370.602, Z    +0.000, E1   +10.342, E3 +97149.585}
SPL {X  -165.650, Y  +380.417, Z    +0.000, E1    +0.167, E3 +97148.501}
SPL {X  -165.650, Y  +381.832, Z    +0.000, E1    -2.686, E3 +97147.927}
SPL {X  -165.650, Y  +385.053, Z    +0.000, E1   -10.073, E3 +97147.832}
SPL {X  -165.650, Y  +388.847, Z    +0.000, E1   -19.524, E3 +97147.796}
SPL {X  -165.650, Y  +393.562, Z    +0.000, E1   -31.212, E3 +97147.280}
SPL {X  -165.650, Y  +400.090, Z    +0.000, E1   -44.561, E3 +97147.135}
SPL {X  -165.650, Y  +415.429, Z    +0.000, E1   -64.815, E3 +97145.193}
SPL {X  -165.650, Y  +470.008, Z    +0.000, E1   -77.011, E3 +97153.737}
SPL {X  -160.882, Y  +714.957, Z    +0.000, E1   -77.470, E3 +97237.443}
ENDSPLINE

SPLINE
SPL {X  -164.302, Y  +696.586, Z    +0.000, E1   -74.218, E3 +97264.105}
ENDSPLINE

SPLINE
SPL {X  -160.977, Y  +714.570, Z    +0.000, E1   -74.086, E3 +97276.017}
SPL {X  -156.453, Y  +729.928, Z    +0.000, E1   -73.507, E3 +97290.584}
SPL {X  -152.193, Y  +740.900, Z    +0.000, E1   -73.135, E3 +97300.150}
SPL {X  -148.880, Y  +748.126, Z    +0.000, E1   -72.716, E3 +97307.932}
SPL {X  -144.434, Y  +756.610, Z    +0.000, E1   -72.338, E3 +97315.782}
SPL {X  -141.532, Y  +761.573, Z    +0.000, E1   -71.800, E3 +97322.422}
SPL {X  -138.580, Y  +766.249, Z    +0.000, E1   -71.449, E3 +97327.484}
SPL {X  -134.851, Y  +771.704, Z    +0.000, E1   -71.081, E3 +97332.879}
SPL {X  -131.668, Y  +776.015, Z    +0.000, E1   -70.566, E3 +97338.153}
SPL {X  -128.114, Y  +780.508, Z    +0.000, E1   -70.155, E3 +97342.748}
SPL {X  -123.825, Y  +785.533, Z    +0.000, E1   -70.642, E3 +97343.496}
SPL {X  -111.068, Y  +798.397, Z    +0.000, E1   -72.944, E3 +97340.940}
SPL {X   -54.368, Y  +831.974, Z    +0.000, E1   -57.152, E3 +97492.823}
ENDSPLINE

SPLINE
SPL {X  -111.514, Y  +797.993, Z    +0.000, E1   -63.064, E3 +97678.954}
SPL {X  -140.675, Y  +762.967, Z    +0.000, E1   -56.489, E3 +97684.917}
SPL {X  -155.138, Y  +733.569, Z    +0.000, E1   -46.550, E3 +97687.221}
SPL {X  -161.585, Y  +711.971, Z    +0.000, E1   -34.503, E3 +97686.271}
SPL {X  -164.796, Y  +692.295, Z    +0.000, E1   -19.289, E3 +97686.306}
SPL {X  -165.632, Y  +677.938, Z    +0.000, E1    -5.073, E3 +97685.677}
SPL {X  -165.650, Y  +673.500, Z    +0.000, E1    +0.000, E3 +97684.711}
SPL {X  -165.650, Y  +671.349, Z    +0.000, E1    +4.619, E3 +97684.216}
SPL {X  -165.650, Y  +666.568, Z    +0.000, E1   +16.799, E3 +97684.091}
SPL {X  -165.650, Y  +661.246, Z    +0.000, E1   +30.569, E3 +97683.871}
SPL {X  -165.650, Y  +652.403, Z    +0.000, E1   +48.665, E3 +97683.510}
SPL {X  -165.650, Y  +637.100, Z    +0.000, E1   +69.106, E3 +97679.850}
SPL {X  -165.650, Y  +616.344, Z    +0.000, E1   +74.941, E3 +97683.099}
SPL {X  -165.650, Y  +575.817, Z    +0.000, E1   +77.800, E3 +97692.028}
SPL {X  -162.613, Y  +346.923, Z    +0.000, E1   +78.263, E3 +97763.701}
SPL {X  -161.207, Y  +340.393, Z    +0.000, E1   +75.705, E3 +97793.564}
SPL {X  -146.302, Y  +300.811, Z    +0.000, E1   +78.008, E3 +97784.445}
ENDSPLINE

SPLINE
SPL {X  -147.825, Y  +303.750, Z    +0.000, E1   +76.548, E3 +97798.877}
SPL {X  -148.167, Y  +304.430, Z    +0.000, E1   +75.276, E3 +97810.970}
ENDSPLINE

SPLINE
SPL {X  -146.983, Y  +302.107, Z    +0.000, E1   +74.473, E3 +97819.451}
SPL {X  -146.624, Y  +301.420, Z    +0.000, E1   +73.294, E3 +97829.935}
SPL {X  -144.830, Y  +298.101, Z    +0.000, E1   +72.333, E3 +97839.458}
SPL {X  -140.483, Y  +290.724, Z    +0.000, E1   +71.922, E3 +97846.616}
SPL {X  -136.362, Y  +284.451, Z    +0.000, E1   +71.514, E3 +97852.782}
SPL {X  -132.604, Y  +279.221, Z    +0.000, E1   +70.988, E3 +97858.810}
SPL {X  -129.663, Y  +275.410, Z    +0.000, E1   +70.632, E3 +97862.734}
SPL {X  -127.149, Y  +272.325, Z    +0.000, E1   +70.073, E3 +97867.114}
SPL {X  -123.924, Y  +268.578, Z    +0.000, E1   +70.633, E3 +97866.931}
SPL {X  -115.163, Y  +259.431, Z    +0.000, E1   +74.058, E3 +97858.040}
SPL {X   -55.479, Y  +222.417, Z    +0.000, E1   +56.403, E3 +98043.894}
ENDSPLINE

SPLINE
SPL {X  -130.757, Y  +276.802, Z    +0.000, E1   +58.343, E3 +98199.830}
SPL {X  -154.788, Y  +319.502, Z    +0.000, E1   +45.389, E3 +98204.029}
SPL {X  -161.887, Y  +343.393, Z    +0.000, E1   +32.461, E3 +98204.485}
SPL {X  -164.949, Y  +363.277, Z    +0.000, E1   +17.059, E3 +98203.760}
SPL {X  -165.638, Y  +376.493, Z    +0.000, E1    +4.395, E3 +98203.398}
SPL {X  -165.650, Y  +380.500, Z    +0.000, E1    +0.000, E3 +98202.509}
SPL {X  -165.650, Y  +381.832, Z    +0.000, E1    -2.686, E3 +98201.981}
SPL {X  -165.650, Y  +385.053, Z    +0.000, E1   -10.073, E3 +98201.886}
SPL {X  -165.650, Y  +388.847, Z    +0.000, E1   -19.524, E3 +98201.851}
SPL {X  -165.650, Y  +393.562, Z    +0.000, E1   -31.212, E3 +98201.334}
SPL {X  -165.650, Y  +400.090, Z    +0.000, E1   -44.561, E3 +98201.189}
SPL {X  -165.650, Y  +415.429, Z    +0.000, E1   -64.815, E3 +98199.248}
SPL {X  -165.650, Y  +470.008, Z    +0.000, E1   -77.011, E3 +98207.791}
SPL {X  -161.095, Y  +714.078, Z    +0.000, E1   -78.221, E3 +98283.327}
ENDSPLINE

SPLINE
SPL {X  -163.418, Y  +702.603, Z    +0.000, E1   -74.313, E3 +98320.722}
ENDSPLINE

SPLINE
SPL {X  -160.284, Y  +717.322, Z    +0.000, E1   -73.988, E3 +98332.486}
SPL {X  -156.453, Y  +729.928, Z    +0.000, E1   -73.507, E3 +98344.638}
SPL {X  -152.193, Y  +740.900, Z    +0.000, E1   -73.135, E3 +98354.205}
SPL {X  -148.880, Y  +748.126, Z    +0.000, E1   -72.716, E3 +98361.986}
SPL {X  -145.823, Y  +754.085, Z    +0.000, E1   -72.288, E3 +98368.757}
SPL {X  -141.906, Y  +760.955, Z    +0.000, E1   -72.057, E3 +98374.448}
SPL {X  -138.580, Y  +766.249, Z    +0.000, E1   -71.449, E3 +98381.538}
SPL {X  -134.851, Y  +771.704, Z    +0.000, E1   -71.081, E3 +98386.933}
SPL {X  -131.668, Y  +776.015, Z    +0.000, E1   -70.566, E3 +98392.207}
SPL {X  -128.114, Y  +780.508, Z    +0.000, E1   -70.155, E3 +98396.802}
SPL {X  -123.825, Y  +785.533, Z    +0.000, E1   -70.642, E3 +98397.550}
SPL {X  -111.068, Y  +798.397, Z    +0.000, E1   -72.944, E3 +98394.994}
SPL {X   -54.135, Y  +832.054, Z    +0.000, E1   -56.519, E3 +98571.013}
ENDSPLINE

SPLINE
SPL {X  -119.915, Y  +789.781, Z    +0.000, E1   -62.637, E3 +98738.629}
SPL {X  -140.675, Y  +762.967, Z    +0.000, E1   -56.489, E3 +98738.971}
SPL {X  -155.138, Y  +733.569, Z    +0.000, E1   -46.550, E3 +98741.275}
SPL {X  -161.585, Y  +711.971, Z    +0.000, E1   -34.503, E3 +98740.325}
SPL {X  -164.796, Y  +692.295, Z    +0.000, E1   -19.289, E3 +98740.360}
SPL {X  -165.632, Y  +677.938, Z    +0.000, E1    -5.073, E3 +98739.731}
SPL {X  -165.650, Y  +673.500, Z    +0.000, E1    +0.000, E3 +98738.765}
SPL {X  -165.650, Y  +671.349, Z    +0.000, E1    +4.619, E3 +98738.270}
SPL {X  -165.650, Y  +666.568, Z    +0.000, E1   +16.799, E3 +98738.145}
SPL {X  -165.650, Y  +661.246, Z    +0.000, E1   +30.569, E3 +98737.925}
SPL {X  -165.650, Y  +652.403, Z    +0.000, E1   +48.665, E3 +98737.564}
SPL {X  -165.650, Y  +637.100, Z    +0.000, E1   +69.106, E3 +98733.904}
SPL {X  -165.650, Y  +616.344, Z    +0.000, E1   +74.941, E3 +98737.154}
SPL {X  -165.650, Y  +575.817, Z    +0.000, E1   +77.800, E3 +98746.083}
SPL {X  -161.405, Y  +341.238, Z    +0.000, E1   +76.606, E3 +98837.382}
SPL {X  -146.302, Y  +300.811, Z    +0.000, E1   +78.008, E3 +98838.499}
ENDSPLINE

SPLINE
SPL {X  -147.825, Y  +303.750, Z    +0.000, E1   +76.548, E3 +98852.931}
SPL {X  -148.167, Y  +304.430, Z    +0.000, E1   +75.276, E3 +98865.024}
ENDSPLINE

SPLINE
SPL {X  -146.983, Y  +302.107, Z    +0.000, E1   +74.473, E3 +98873.505}
SPL {X  -146.624, Y  +301.420, Z    +0.000, E1   +73.294, E3 +98883.989}
SPL {X  -144.830, Y  +298.101, Z    +0.000, E1   +72.333, E3 +98893.512}
SPL {X  -140.483, Y  +290.724, Z    +0.000, E1   +71.922, E3 +98900.670}
SPL {X  -136.362, Y  +284.451, Z    +0.000, E1   +71.514, E3 +98906.836}
SPL {X  -132.604, Y  +279.221, Z    +0.000, E1   +70.988, E3 +98912.865}
SPL {X  -129.663, Y  +275.410, Z    +0.000, E1   +70.632, E3 +98916.788}
SPL {X  -127.149, Y  +272.325, Z    +0.000, E1   +70.073, E3 +98921.168}
SPL {X  -123.924, Y  +268.578, Z    +0.000, E1   +70.633, E3 +98920.985}
SPL {X  -115.163, Y  +259.431, Z    +0.000, E1   +74.058, E3 +98912.094}
SPL {X   -55.479, Y  +222.417, Z    +0.000, E1   +56.403, E3 +99097.948}
ENDSPLINE

SPLINE
SPL {X  -130.757, Y  +276.802, Z    +0.000, E1   +58.343, E3 +99253.884}
SPL {X  -157.227, Y  +326.349, Z    +0.000, E1   +42.092, E3 +99257.530}
SPL {X  -163.771, Y  +353.623, Z    +0.000, E1   +25.144, E3 +99258.743}
SPL {X  -165.462, Y  +370.602, Z    +0.000, E1   +10.342, E3 +99257.693}
SPL {X  -165.650, Y  +380.752, Z    +0.000, E1    -0.182, E3 +99256.473}
SPL {X  -165.650, Y  +385.053, Z    +0.000, E1   -10.073, E3 +99255.940}
SPL {X  -165.650, Y  +388.847, Z    +0.000, E1   -19.524, E3 +99255.905}
SPL {X  -165.650, Y  +393.562, Z    +0.000, E1   -31.212, E3 +99255.388}
SPL {X  -165.650, Y  +400.090, Z    +0.000, E1   -44.561, E3 +99255.243}
SPL {X  -165.650, Y  +415.429, Z    +0.000, E1   -64.815, E3 +99253.302}
SPL {X  -165.650, Y  +470.008, Z    +0.000, E1   -77.011, E3 +99261.846}
SPL {X  -160.882, Y  +714.957, Z    +0.000, E1   -77.470, E3 +99345.551}
ENDSPLINE

SPLINE
SPL {X  -164.302, Y  +696.586, Z    +0.000, E1   -74.218, E3 +99372.213}
ENDSPLINE

SPLINE
SPL {X  -160.977, Y  +714.570, Z    +0.000, E1   -74.086, E3 +99384.125}
SPL {X  -156.453, Y  +729.928, Z    +0.000, E1   -73.507, E3 +99398.692}
SPL {X  -152.193, Y  +740.900, Z    +0.000, E1   -73.135, E3 +99408.259}
SPL {X  -148.880, Y  +748.126, Z    +0.000, E1   -72.716, E3 +99416.040}
SPL {X  -145.823, Y  +754.085, Z    +0.000, E1   -72.288, E3 +99422.811}
SPL {X  -141.906, Y  +760.955, Z    +0.000, E1   -72.057, E3 +99428.502}
SPL {X  -138.580, Y  +766.249, Z    +0.000, E1   -71.449, E3 +99435.592}
SPL {X  -134.851, Y  +771.704, Z    +0.000, E1   -71.081, E3 +99440.987}
SPL {X  -130.513, Y  +777.511, Z    +0.000, E1   -70.561, E3 +99447.169}
SPL {X  -127.002, Y  +781.850, Z    +0.000, E1   -69.819, E3 +99453.024}
SPL {X  -121.778, Y  +787.794, Z    +0.000, E1   -71.623, E3 +99449.073}
SPL {X  -111.068, Y  +798.397, Z    +0.000, E1   -72.944, E3 +99449.048}
SPL {X   -54.368, Y  +831.974, Z    +0.000, E1   -57.152, E3 +99600.931}
ENDSPLINE

SPLINE
SPL {X  -111.514, Y  +797.993, Z    +0.000, E1   -63.064, E3 +99787.062}
SPL {X  -140.675, Y  +762.967, Z    +0.000, E1   -56.489, E3 +99793.025}
SPL {X  -155.138, Y  +733.569, Z    +0.000, E1   -46.550, E3 +99795.329}
SPL {X  -161.585, Y  +711.971, Z    +0.000, E1   -34.503, E3 +99794.380}
SPL {X  -164.796, Y  +692.295, Z    +0.000, E1   -19.289, E3 +99794.414}
SPL {X  -165.632, Y  +677.938, Z    +0.000, E1    -5.073, E3 +99793.785}
SPL {X  -165.650, Y  +673.500, Z    +0.000, E1    +0.000, E3 +99792.819}
SPL {X  -165.650, Y  +671.349, Z    +0.000, E1    +4.619, E3 +99792.324}
SPL {X  -165.650, Y  +666.568, Z    +0.000, E1   +16.799, E3 +99792.199}
SPL {X  -165.650, Y  +661.246, Z    +0.000, E1   +30.569, E3 +99791.980}
SPL {X  -165.650, Y  +652.403, Z    +0.000, E1   +48.665, E3 +99791.618}
SPL {X  -165.650, Y  +637.100, Z    +0.000, E1   +69.106, E3 +99787.958}
SPL {X  -165.650, Y  +616.344, Z    +0.000, E1   +74.941, E3 +99791.208}
SPL {X  -165.650, Y  +575.817, Z    +0.000, E1   +77.800, E3 +99800.137}
SPL {X  -161.405, Y  +341.238, Z    +0.000, E1   +76.606, E3 +99891.436}
SPL {X  -146.302, Y  +300.811, Z    +0.000, E1   +78.008, E3 +99892.553}
ENDSPLINE

SPLINE
SPL {X  -147.825, Y  +303.750, Z    +0.000, E1   +76.548, E3 +99906.986}
SPL {X  -148.167, Y  +304.430, Z    +0.000, E1   +75.276, E3 +99919.078}
ENDSPLINE

SPLINE
SPL {X  -146.983, Y  +302.107, Z    +0.000, E1   +74.473, E3 +99927.559}
SPL {X  -146.624, Y  +301.420, Z    +0.000, E1   +73.294, E3 +99938.043}
SPL {X  -144.830, Y  +298.101, Z    +0.000, E1   +72.333, E3 +99947.567}
SPL {X  -140.980, Y  +291.526, Z    +0.000, E1   +72.160, E3 +99952.492}
SPL {X  -137.379, Y  +285.943, Z    +0.000, E1   +71.537, E3 +99959.946}
SPL {X  -133.329, Y  +280.198, Z    +0.000, E1   +71.389, E3 +99963.975}
SPL {X  -130.835, Y  +276.902, Z    +0.000, E1   +70.642, E3 +99969.971}
SPL {X  -127.149, Y  +272.325, Z    +0.000, E1   +70.073, E3 +99975.222}
SPL {X  -123.924, Y  +268.578, Z    +0.000, E1   +70.633, E3 +99975.039}
SPL {X  -115.163, Y  +259.431, Z    +0.000, E1   +74.058, E3 +99966.148}
SPL {X   -55.479, Y  +222.417, Z    +0.000, E1   +56.403, E3 +100152.002}
ENDSPLINE

SPLINE
SPL {X  -130.757, Y  +276.802, Z    +0.000, E1   +58.343, E3 +100307.938}
SPL {X  -154.788, Y  +319.502, Z    +0.000, E1   +45.389, E3 +100312.137}
SPL {X  -161.887, Y  +343.393, Z    +0.000, E1   +32.461, E3 +100312.593}
SPL {X  -164.949, Y  +363.277, Z    +0.000, E1   +17.059, E3 +100311.868}
SPL {X  -165.638, Y  +376.493, Z    +0.000, E1    +4.395, E3 +100311.507}
SPL {X  -165.650, Y  +380.500, Z    +0.000, E1    +0.000, E3 +100310.617}
SPL {X  -165.650, Y  +381.832, Z    +0.000, E1    -2.686, E3 +100310.089}
SPL {X  -165.650, Y  +385.053, Z    +0.000, E1   -10.073, E3 +100309.994}
SPL {X  -165.650, Y  +388.847, Z    +0.000, E1   -19.524, E3 +100309.959}
SPL {X  -165.650, Y  +393.562, Z    +0.000, E1   -31.212, E3 +100309.443}
SPL {X  -165.650, Y  +400.090, Z    +0.000, E1   -44.561, E3 +100309.297}
SPL {X  -165.650, Y  +415.429, Z    +0.000, E1   -64.815, E3 +100307.356}
SPL {X  -165.650, Y  +470.008, Z    +0.000, E1   -77.011, E3 +100315.900}
SPL {X  -160.882, Y  +714.957, Z    +0.000, E1   -77.470, E3 +100399.605}
ENDSPLINE

SPLINE
SPL {X  -164.302, Y  +696.586, Z    +0.000, E1   -74.218, E3 +100426.267}
ENDSPLINE

SPLINE
SPL {X  -160.977, Y  +714.570, Z    +0.000, E1   -74.086, E3 +100438.179}
SPL {X  -156.453, Y  +729.928, Z    +0.000, E1   -73.507, E3 +100452.746}
SPL {X  -152.193, Y  +740.900, Z    +0.000, E1   -73.135, E3 +100462.313}
SPL {X  -148.880, Y  +748.126, Z    +0.000, E1   -72.716, E3 +100470.094}
SPL {X  -144.434, Y  +756.610, Z    +0.000, E1   -72.338, E3 +100477.944}
SPL {X  -141.532, Y  +761.573, Z    +0.000, E1   -71.800, E3 +100484.584}
SPL {X  -138.580, Y  +766.249, Z    +0.000, E1   -71.449, E3 +100489.646}
SPL {X  -134.851, Y  +771.704, Z    +0.000, E1   -71.081, E3 +100495.041}
SPL {X  -131.668, Y  +776.015, Z    +0.000, E1   -70.566, E3 +100500.315}
SPL {X  -128.114, Y  +780.508, Z    +0.000, E1   -70.155, E3 +100504.910}
SPL {X  -125.843, Y  +783.219, Z    +0.000, E1   -69.779, E3 +100508.014}
SPL {X  -118.977, Y  +790.758, Z    +0.000, E1   -71.976, E3 +100503.196}
SPL {X   -54.135, Y  +832.054, Z    +0.000, E1   -56.519, E3 +100679.121}
ENDSPLINE

SPLINE
SPL {X  -119.915, Y  +789.781, Z    +0.000, E1   -62.637, E3 +100846.737}
SPL {X  -140.675, Y  +762.967, Z    +0.000, E1   -56.489, E3 +100847.079}
SPL {X  -155.138, Y  +733.569, Z    +0.000, E1   -46.550, E3 +100849.383}
SPL {X  -161.585, Y  +711.971, Z    +0.000, E1   -34.503, E3 +100848.434}
SPL {X  -164.796, Y  +692.295, Z    +0.000, E1   -19.289, E3 +100848.468}
SPL {X  -165.571, Y  +680.631, Z    +0.000, E1    -7.833, E3 +100847.915}
SPL {X  -165.650, Y  +673.591, Z    +0.000, E1    -0.194, E3 +100846.919}
SPL {X  -165.650, Y  +671.349, Z    +0.000, E1    +4.619, E3 +100846.378}
SPL {X  -165.650, Y  +666.568, Z    +0.000, E1   +16.799, E3 +100846.254}
SPL {X  -165.650, Y  +661.246, Z    +0.000, E1   +30.569, E3 +100846.034}
SPL {X  -165.650, Y  +655.398, Z    +0.000, E1   +43.871, E3 +100845.481}
SPL {X  -165.650, Y  +646.168, Z    +0.000, E1   +58.442, E3 +100844.576}
SPL {X  -165.650, Y  +629.125, Z    +0.000, E1   +72.389, E3 +100842.873}
SPL {X  -165.650, Y  +575.817, Z    +0.000, E1   +77.800, E3 +100854.191}
SPL {X  -161.405, Y  +341.238, Z    +0.000, E1   +76.606, E3 +100945.490}
SPL {X  -146.302, Y  +300.811, Z    +0.000, E1   +78.008, E3 +100946.607}
ENDSPLINE

SPLINE
SPL {X  -147.825, Y  +303.750, Z    +0.000, E1   +76.548, E3 +100961.040}
SPL {X  -148.167, Y  +304.430, Z    +0.000, E1   +75.276, E3 +100973.132}
ENDSPLINE

SPLINE
SPL {X  -146.983, Y  +302.107, Z    +0.000, E1   +74.473, E3 +100981.613}
SPL {X  -146.624, Y  +301.420, Z    +0.000, E1   +73.294, E3 +100992.097}
SPL {X  -144.830, Y  +298.101, Z    +0.000, E1   +72.333, E3 +101001.621}
SPL {X  -140.980, Y  +291.526, Z    +0.000, E1   +72.160, E3 +101006.546}
SPL {X  -137.379, Y  +285.943, Z    +0.000, E1   +71.537, E3 +101014.001}
SPL {X  -133.329, Y  +280.198, Z    +0.000, E1   +71.389, E3 +101018.029}
SPL {X  -130.835, Y  +276.902, Z    +0.000, E1   +70.642, E3 +101024.025}
SPL {X  -127.149, Y  +272.325, Z    +0.000, E1   +70.073, E3 +101029.276}
SPL {X  -123.924, Y  +268.578, Z    +0.000, E1   +70.633, E3 +101029.093}
SPL {X  -115.163, Y  +259.431, Z    +0.000, E1   +74.058, E3 +101020.202}
SPL {X   -55.479, Y  +222.417, Z    +0.000, E1   +56.403, E3 +101206.056}
ENDSPLINE

SPLINE
SPL {X  -130.757, Y  +276.802, Z    +0.000, E1   +58.343, E3 +101361.993}
SPL {X  -154.788, Y  +319.502, Z    +0.000, E1   +45.389, E3 +101366.191}
SPL {X  -161.887, Y  +343.393, Z    +0.000, E1   +32.461, E3 +101366.647}
SPL {X  -164.949, Y  +363.277, Z    +0.000, E1   +17.059, E3 +101365.922}
SPL {X  -165.638, Y  +376.493, Z    +0.000, E1    +4.395, E3 +101365.561}
SPL {X  -165.650, Y  +380.500, Z    +0.000, E1    +0.000, E3 +101364.671}
SPL {X  -165.650, Y  +381.832, Z    +0.000, E1    -2.686, E3 +101364.143}
SPL {X  -165.650, Y  +385.053, Z    +0.000, E1   -10.073, E3 +101364.048}
SPL {X  -165.650, Y  +388.847, Z    +0.000, E1   -19.524, E3 +101364.013}
SPL {X  -165.650, Y  +393.562, Z    +0.000, E1   -31.212, E3 +101363.497}
SPL {X  -165.650, Y  +400.090, Z    +0.000, E1   -44.561, E3 +101363.351}
SPL {X  -165.650, Y  +415.429, Z    +0.000, E1   -64.815, E3 +101361.410}
SPL {X  -165.650, Y  +470.008, Z    +0.000, E1   -77.011, E3 +101369.954}
SPL {X  -160.882, Y  +714.957, Z    +0.000, E1   -77.470, E3 +101453.659}
ENDSPLINE

SPLINE
SPL {X  -164.302, Y  +696.586, Z    +0.000, E1   -74.218, E3 +101480.321}
ENDSPLINE

SPLINE
SPL {X  -160.977, Y  +714.570, Z    +0.000, E1   -74.086, E3 +101492.233}
SPL {X  -156.453, Y  +729.928, Z    +0.000, E1   -73.507, E3 +101506.800}
SPL {X  -152.193, Y  +740.900, Z    +0.000, E1   -73.135, E3 +101516.367}
SPL {X  -148.880, Y  +748.126, Z    +0.000, E1   -72.716, E3 +101524.148}
SPL {X  -144.434, Y  +756.610, Z    +0.000, E1   -72.338, E3 +101531.998}
SPL {X  -141.532, Y  +761.573, Z    +0.000, E1   -71.800, E3 +101538.638}
SPL {X  -138.580, Y  +766.249, Z    +0.000, E1   -71.449, E3 +101543.700}
SPL {X  -134.851, Y  +771.704, Z    +0.000, E1   -71.081, E3 +101549.095}
SPL {X  -131.668, Y  +776.015, Z    +0.000, E1   -70.566, E3 +101554.369}
SPL {X  -128.114, Y  +780.508, Z    +0.000, E1   -70.155, E3 +101558.964}
SPL {X  -125.843, Y  +783.219, Z    +0.000, E1   -69.779, E3 +101562.068}
SPL {X  -118.977, Y  +790.758, Z    +0.000, E1   -71.976, E3 +101557.250}
SPL {X   -54.135, Y  +832.054, Z    +0.000, E1   -56.519, E3 +101733.175}
ENDSPLINE

SPLINE
SPL {X  -119.915, Y  +789.781, Z    +0.000, E1   -62.637, E3 +101900.791}
SPL {X  -140.675, Y  +762.967, Z    +0.000, E1   -56.489, E3 +101901.133}
SPL {X  -155.138, Y  +733.569, Z    +0.000, E1   -46.550, E3 +101903.437}
SPL {X  -161.585, Y  +711.971, Z    +0.000, E1   -34.503, E3 +101902.488}
SPL {X  -164.796, Y  +692.295, Z    +0.000, E1   -19.289, E3 +101902.522}
SPL {X  -165.571, Y  +680.631, Z    +0.000, E1    -7.833, E3 +101901.969}
SPL {X  -165.650, Y  +673.591, Z    +0.000, E1    -0.194, E3 +101900.973}
SPL {X  -165.650, Y  +671.349, Z    +0.000, E1    +4.619, E3 +101900.432}
SPL {X  -165.650, Y  +666.568, Z    +0.000, E1   +16.799, E3 +101900.308}
SPL {X  -165.650, Y  +661.246, Z    +0.000, E1   +30.569, E3 +101900.088}
SPL {X  -165.650, Y  +655.398, Z    +0.000, E1   +43.871, E3 +101899.535}
SPL {X  -165.650, Y  +646.168, Z    +0.000, E1   +58.442, E3 +101898.630}
SPL {X  -165.650, Y  +629.125, Z    +0.000, E1   +72.389, E3 +101896.927}
SPL {X  -165.650, Y  +575.817, Z    +0.000, E1   +77.800, E3 +101908.245}
SPL {X  -161.405, Y  +341.238, Z    +0.000, E1   +76.606, E3 +101999.545}
SPL {X  -146.302, Y  +300.811, Z    +0.000, E1   +78.008, E3 +102000.661}
ENDSPLINE

SPLINE
SPL {X  -147.825, Y  +303.750, Z    +0.000, E1   +76.548, E3 +102015.094}
SPL {X  -148.167, Y  +304.430, Z    +0.000, E1   +75.276, E3 +102027.186}
ENDSPLINE

SPLINE
SPL {X  -146.983, Y  +302.107, Z    +0.000, E1   +74.473, E3 +102035.667}
SPL {X  -146.624, Y  +301.420, Z    +0.000, E1   +73.294, E3 +102046.151}
SPL {X  -144.830, Y  +298.101, Z    +0.000, E1   +72.333, E3 +102055.675}
SPL {X  -140.980, Y  +291.526, Z    +0.000, E1   +72.160, E3 +102060.600}
SPL {X  -137.379, Y  +285.943, Z    +0.000, E1   +71.537, E3 +102068.055}
SPL {X  -133.329, Y  +280.198, Z    +0.000, E1   +71.389, E3 +102072.083}
SPL {X  -130.835, Y  +276.902, Z    +0.000, E1   +70.642, E3 +102078.079}
SPL {X  -127.149, Y  +272.325, Z    +0.000, E1   +70.073, E3 +102083.331}
SPL {X  -123.924, Y  +268.578, Z    +0.000, E1   +70.633, E3 +102083.147}
SPL {X  -115.163, Y  +259.431, Z    +0.000, E1   +74.058, E3 +102074.256}
SPL {X   -55.479, Y  +222.417, Z    +0.000, E1   +56.403, E3 +102260.110}
ENDSPLINE

SPLINE
SPL {X  -130.757, Y  +276.802, Z    +0.000, E1   +58.343, E3 +102416.047}
SPL {X  -154.788, Y  +319.502, Z    +0.000, E1   +45.389, E3 +102420.245}
SPL {X  -161.887, Y  +343.393, Z    +0.000, E1   +32.461, E3 +102420.701}
SPL {X  -164.949, Y  +363.277, Z    +0.000, E1   +17.059, E3 +102419.976}
SPL {X  -165.638, Y  +376.493, Z    +0.000, E1    +4.395, E3 +102419.615}
SPL {X  -165.650, Y  +380.500, Z    +0.000, E1    +0.000, E3 +102418.725}
SPL {X  -165.650, Y  +381.832, Z    +0.000, E1    -2.686, E3 +102418.197}
SPL {X  -165.650, Y  +385.053, Z    +0.000, E1   -10.073, E3 +102418.102}
SPL {X  -165.650, Y  +388.847, Z    +0.000, E1   -19.524, E3 +102418.067}
SPL {X  -165.650, Y  +393.562, Z    +0.000, E1   -31.212, E3 +102417.551}
SPL {X  -165.650, Y  +400.090, Z    +0.000, E1   -44.561, E3 +102417.405}
SPL {X  -165.650, Y  +415.429, Z    +0.000, E1   -64.815, E3 +102415.464}
SPL {X  -165.650, Y  +470.008, Z    +0.000, E1   -77.011, E3 +102424.008}
SPL {X  -160.882, Y  +714.957, Z    +0.000, E1   -77.470, E3 +102507.714}
ENDSPLINE

SPLINE
SPL {X  -164.302, Y  +696.586, Z    +0.000, E1   -74.218, E3 +102534.375}
ENDSPLINE

SPLINE
SPL {X  -160.977, Y  +714.570, Z    +0.000, E1   -74.086, E3 +102546.287}
SPL {X  -156.453, Y  +729.928, Z    +0.000, E1   -73.507, E3 +102560.854}
SPL {X  -152.193, Y  +740.900, Z    +0.000, E1   -73.135, E3 +102570.421}
SPL {X  -148.880, Y  +748.126, Z    +0.000, E1   -72.716, E3 +102578.202}
SPL {X  -144.434, Y  +756.610, Z    +0.000, E1   -72.338, E3 +102586.052}
SPL {X  -141.532, Y  +761.573, Z    +0.000, E1   -71.800, E3 +102592.692}
SPL {X  -138.580, Y  +766.249, Z    +0.000, E1   -71.449, E3 +102597.754}
SPL {X  -134.851, Y  +771.704, Z    +0.000, E1   -71.081, E3 +102603.149}
SPL {X  -131.668, Y  +776.015, Z    +0.000, E1   -70.566, E3 +102608.423}
SPL {X  -128.114, Y  +780.508, Z    +0.000, E1   -70.155, E3 +102613.018}
SPL {X  -125.843, Y  +783.219, Z    +0.000, E1   -69.779, E3 +102616.122}
SPL {X  -118.977, Y  +790.758, Z    +0.000, E1   -71.976, E3 +102611.304}
SPL {X   -54.135, Y  +832.054, Z    +0.000, E1   -56.519, E3 +102787.229}
ENDSPLINE

SPLINE
SPL {X  -119.915, Y  +789.781, Z    +0.000, E1   -62.637, E3 +102954.845}
SPL {X  -140.675, Y  +762.967, Z    +0.000, E1   -56.489, E3 +102955.187}
SPL {X  -155.138, Y  +733.569, Z    +0.000, E1   -46.550, E3 +102957.491}
SPL {X  -161.585, Y  +711.971, Z    +0.000, E1   -34.503, E3 +102956.542}
SPL {X  -164.796, Y  +692.295, Z    +0.000, E1   -19.289, E3 +102956.576}
SPL {X  -165.571, Y  +680.631, Z    +0.000, E1    -7.833, E3 +102956.023}
SPL {X  -165.650, Y  +673.591, Z    +0.000, E1    -0.194, E3 +102955.027}
SPL {X  -165.650, Y  +671.349, Z    +0.000, E1    +4.619, E3 +102954.486}
SPL {X  -165.650, Y  +666.568, Z    +0.000, E1   +16.799, E3 +102954.362}
SPL {X  -165.650, Y  +661.246, Z    +0.000, E1   +30.569, E3 +102954.142}
SPL {X  -165.650, Y  +655.398, Z    +0.000, E1   +43.871, E3 +102953.589}
SPL {X  -165.650, Y  +646.168, Z    +0.000, E1   +58.442, E3 +102952.684}
SPL {X  -165.650, Y  +629.125, Z    +0.000, E1   +72.389, E3 +102950.981}
SPL {X  -165.650, Y  +575.817, Z    +0.000, E1   +77.800, E3 +102962.299}
SPL {X  -161.405, Y  +341.238, Z    +0.000, E1   +76.606, E3 +103053.599}
SPL {X  -146.302, Y  +300.811, Z    +0.000, E1   +78.008, E3 +103054.715}
ENDSPLINE

SPLINE
SPL {X  -147.825, Y  +303.750, Z    +0.000, E1   +76.548, E3 +103069.148}
SPL {X  -148.167, Y  +304.430, Z    +0.000, E1   +75.276, E3 +103081.241}
ENDSPLINE

SPLINE
SPL {X  -146.983, Y  +302.107, Z    +0.000, E1   +74.473, E3 +103089.721}
SPL {X  -146.624, Y  +301.420, Z    +0.000, E1   +73.294, E3 +103100.205}
SPL {X  -144.830, Y  +298.101, Z    +0.000, E1   +72.333, E3 +103109.729}
SPL {X  -140.980, Y  +291.526, Z    +0.000, E1   +72.160, E3 +103114.654}
SPL {X  -137.379, Y  +285.943, Z    +0.000, E1   +71.537, E3 +103122.109}
SPL {X  -133.329, Y  +280.198, Z    +0.000, E1   +71.389, E3 +103126.137}
SPL {X  -130.835, Y  +276.902, Z    +0.000, E1   +70.642, E3 +103132.133}
SPL {X  -127.149, Y  +272.325, Z    +0.000, E1   +70.073, E3 +103137.385}
SPL {X  -123.924, Y  +268.578, Z    +0.000, E1   +70.633, E3 +103137.201}
SPL {X  -115.163, Y  +259.431, Z    +0.000, E1   +74.058, E3 +103128.311}
SPL {X   -55.479, Y  +222.417, Z    +0.000, E1   +56.403, E3 +103314.164}
ENDSPLINE

SPLINE
SPL {X  -130.757, Y  +276.802, Z    +0.000, E1   +58.343, E3 +103470.101}
SPL {X  -154.788, Y  +319.502, Z    +0.000, E1   +45.389, E3 +103474.299}
SPL {X  -161.887, Y  +343.393, Z    +0.000, E1   +32.461, E3 +103474.755}
SPL {X  -164.949, Y  +363.277, Z    +0.000, E1   +17.059, E3 +103474.030}
SPL {X  -165.638, Y  +376.493, Z    +0.000, E1    +4.395, E3 +103473.669}
SPL {X  -165.650, Y  +380.500, Z    +0.000, E1    +0.000, E3 +103472.779}
SPL {X  -165.650, Y  +381.832, Z    +0.000, E1    -2.686, E3 +103472.251}
SPL {X  -165.650, Y  +385.053, Z    +0.000, E1   -10.073, E3 +103472.156}
SPL {X  -165.650, Y  +388.847, Z    +0.000, E1   -19.524, E3 +103472.121}
SPL {X  -165.650, Y  +393.562, Z    +0.000, E1   -31.212, E3 +103471.605}
SPL {X  -165.650, Y  +400.090, Z    +0.000, E1   -44.561, E3 +103471.459}
SPL {X  -165.650, Y  +415.429, Z    +0.000, E1   -64.815, E3 +103469.518}
SPL {X  -165.650, Y  +470.008, Z    +0.000, E1   -77.011, E3 +103478.062}
SPL {X  -160.882, Y  +714.957, Z    +0.000, E1   -77.470, E3 +103561.768}
ENDSPLINE

SPLINE
SPL {X  -163.522, Y  +701.969, Z    +0.000, E1   -74.236, E3 +103591.423}
ENDSPLINE

